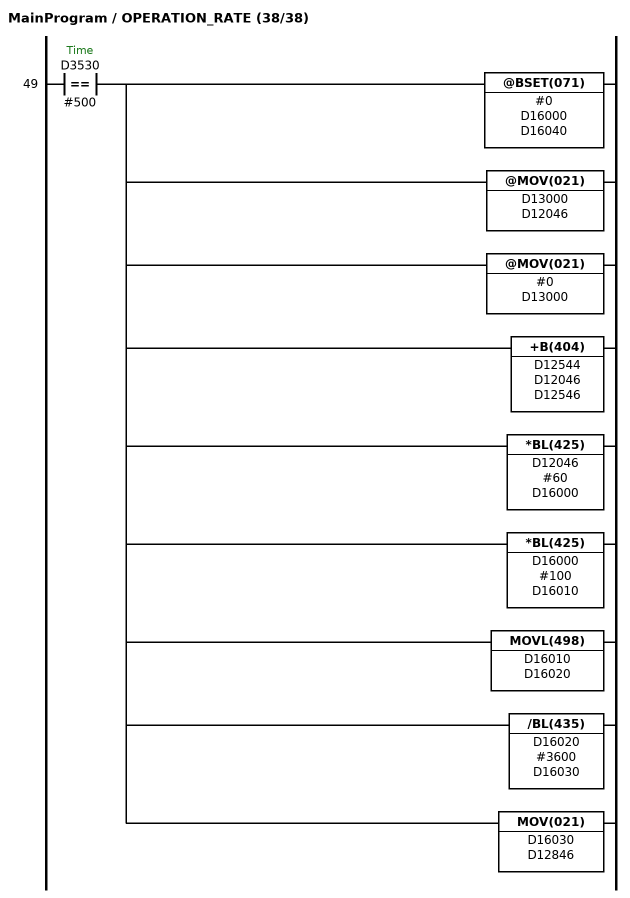
; [picture p288: MainProgram / OPERATION_RATE, rungs 49-49]
; rung 49
LD=L(301) D3530 #500  ; Time
@BSET(071) #0 D16000 D16040
@MOV(021) D13000 D12046
@MOV(021) #0 D13000
+B(404) D12544 D12046 D12546
*BL(425) D12046 #60 D16000
*BL(425) D16000 #100 D16010
MOVL(498) D16010 D16020
/BL(435) D16020 #3600 D16030
MOV(021) D16030 D12846

### Section MASTER_SWITCH_ON

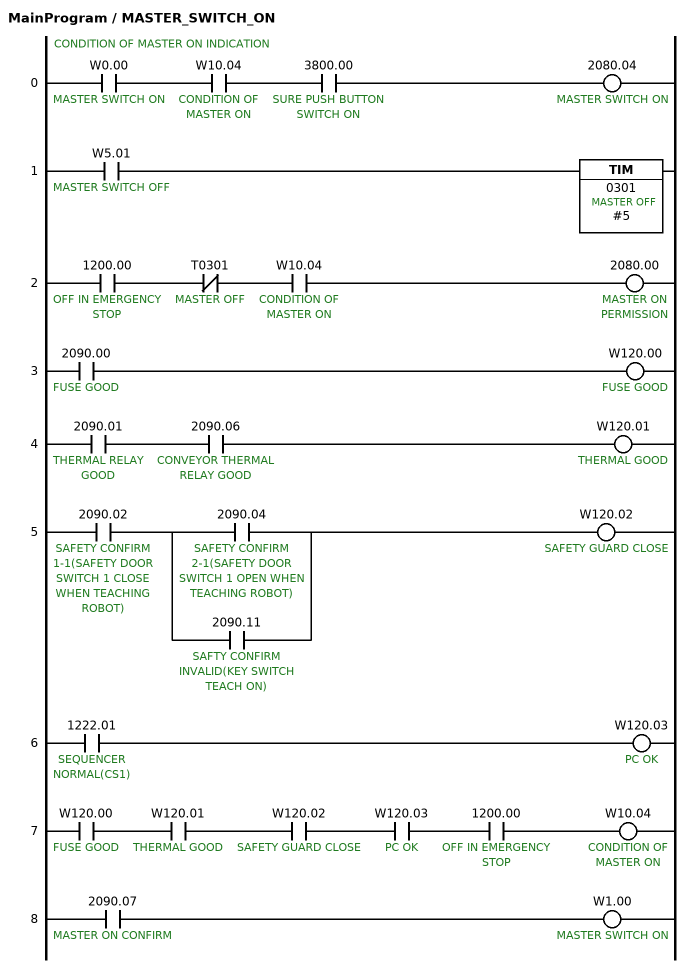
; rung 0: CONDITION OF MASTER ON INDICATION
LD W0.00  ; MASTER SWITCH ON
AND W10.04  ; CONDITION OF MASTER ON
AND 3800.00  ; SURE PUSH BUTTON SWITCH ON
OUT 2080.04  ; MASTER SWITCH ON
; rung 1
LD W5.01  ; MASTER SWITCH OFF
TIM 0301 #5  ; MASTER OFF
; rung 2
LD 1200.00  ; OFF IN EMERGENCY STOP
ANDNOT T0301  ; MASTER OFF
AND W10.04  ; CONDITION OF MASTER ON
OUT 2080.00  ; MASTER ON PERMISSION
; rung 3
LD 2090.00  ; FUSE GOOD
OUT W120.00  ; FUSE GOOD
; rung 4
LD 2090.01  ; THERMAL RELAY GOOD
AND 2090.06  ; CONVEYOR THERMAL RELAY GOOD
OUT W120.01  ; THERMAL GOOD
; rung 5
LD 2090.02  ; SAFETY CONFIRM 1-1(SAFETY DOOR SWITCH 1 CLOSE WHEN TEACHING ROBOT)
LD 2090.04  ; SAFETY CONFIRM 2-1(SAFETY DOOR SWITCH 1 OPEN WHEN TEACHING ROBOT)
OR 2090.11  ; SAFTY CONFIRM INVALID(KEY SWITCH TEACH ON)
ANDLD
OUT W120.02  ; SAFETY GUARD CLOSE
; rung 6
LD 1222.01  ; SEQUENCER NORMAL(CS1)
OUT W120.03  ; PC OK
; rung 7
LD W120.00  ; FUSE GOOD
AND W120.01  ; THERMAL GOOD
AND W120.02  ; SAFETY GUARD CLOSE
AND W120.03  ; PC OK
AND 1200.00  ; OFF IN EMERGENCY STOP
OUT W10.04  ; CONDITION OF MASTER ON
; rung 8
LD 2090.07  ; MASTER ON CONFIRM
OUT W1.00  ; MASTER SWITCH ON

### Section MODE_SELECT

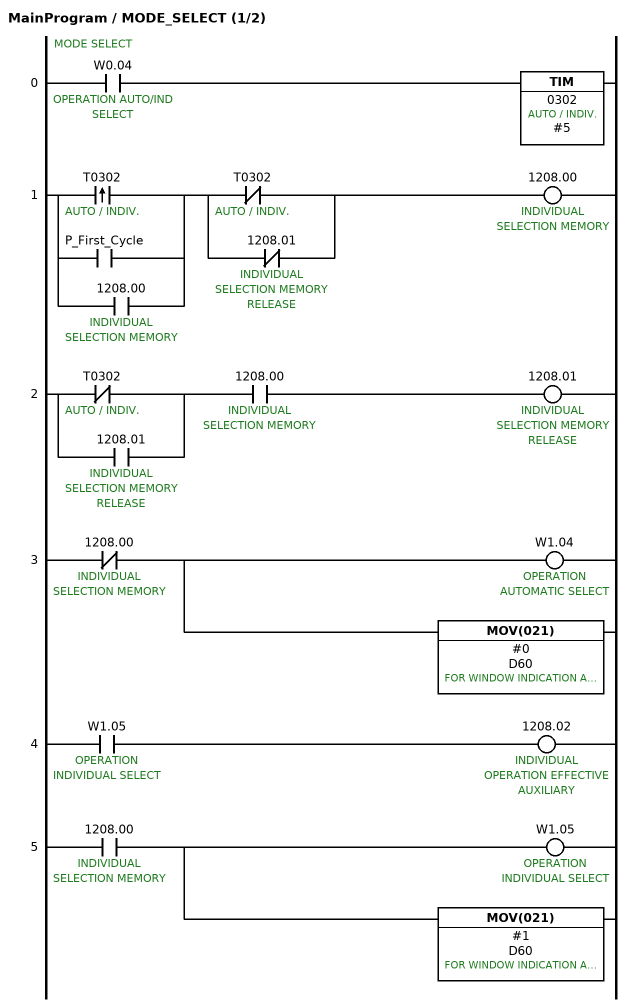
; rung 0: MODE SELECT
LD W0.04  ; OPERATION AUTO/IND SELECT
TIM 0302 #5  ; AUTO / INDIV.
; rung 1
@LD T0302  ; AUTO / INDIV.
OR P_First_Cycle
OR 1208.00  ; INDIVIDUAL SELECTION MEMORY
LDNOT T0302  ; AUTO / INDIV.
ORNOT 1208.01  ; INDIVIDUAL SELECTION MEMORY RELEASE
ANDLD
OUT 1208.00  ; INDIVIDUAL SELECTION MEMORY
; rung 2
LDNOT T0302  ; AUTO / INDIV.
OR 1208.01  ; INDIVIDUAL SELECTION MEMORY RELEASE
AND 1208.00  ; INDIVIDUAL SELECTION MEMORY
OUT 1208.01  ; INDIVIDUAL SELECTION MEMORY RELEASE
; rung 3
LDNOT 1208.00  ; INDIVIDUAL SELECTION MEMORY
OUT W1.04  ; OPERATION AUTOMATIC SELECT
MOV(021) #0 D60  ; FOR WINDOW INDICATION AT INDIVIDUAL
; rung 4
LD W1.05  ; OPERATION INDIVIDUAL SELECT
OUT 1208.02  ; INDIVIDUAL OPERATION EFFECTIVE AUXILIARY
; rung 5
LD 1208.00  ; INDIVIDUAL SELECTION MEMORY
OUT W1.05  ; OPERATION INDIVIDUAL SELECT
MOV(021) #1 D60  ; FOR WINDOW INDICATION AT INDIVIDUAL

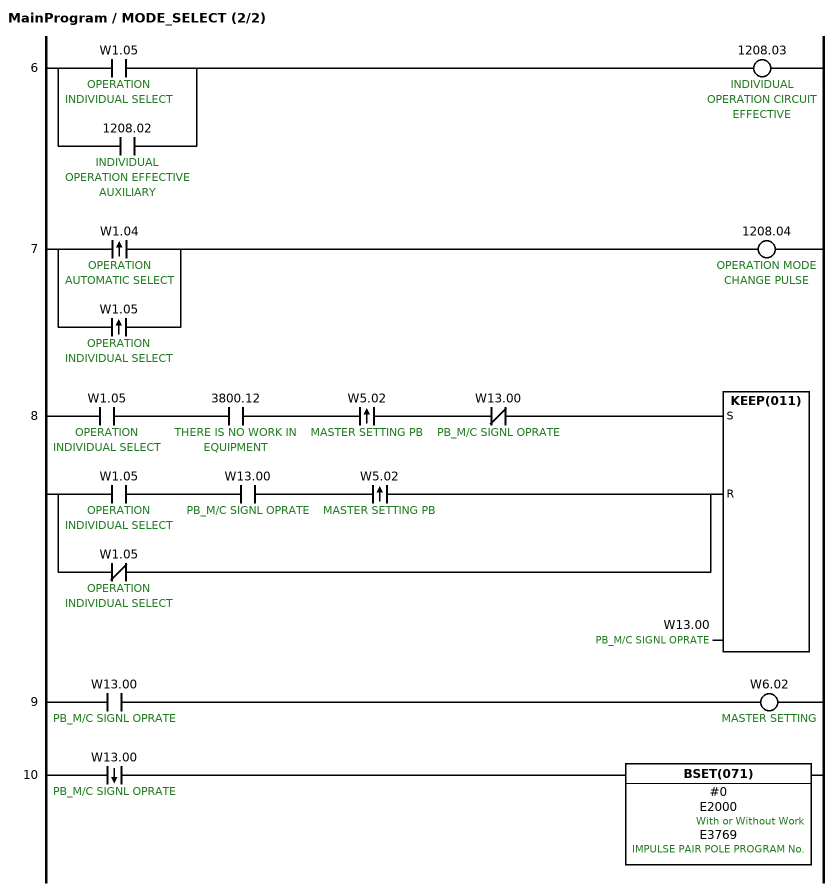
; rung 6
LD W1.05  ; OPERATION INDIVIDUAL SELECT
OR 1208.02  ; INDIVIDUAL OPERATION EFFECTIVE AUXILIARY
OUT 1208.03  ; INDIVIDUAL OPERATION CIRCUIT EFFECTIVE
; rung 7
@LD W1.04  ; OPERATION AUTOMATIC SELECT
@OR W1.05  ; OPERATION INDIVIDUAL SELECT
OUT 1208.04  ; OPERATION MODE CHANGE PULSE
; rung 8
LD W1.05  ; OPERATION INDIVIDUAL SELECT
AND 3800.12  ; THERE IS NO WORK IN EQUIPMENT
@AND W5.02  ; MASTER SETTING PB
ANDNOT W13.00  ; PB_M/C SIGNL OPRATE
LD W1.05  ; OPERATION INDIVIDUAL SELECT
AND W13.00  ; PB_M/C SIGNL OPRATE
@AND W5.02  ; MASTER SETTING PB
ORNOT W1.05  ; OPERATION INDIVIDUAL SELECT
KEEP(011) W13.00  ; PB_M/C SIGNL OPRATE
; rung 9
LD W13.00  ; PB_M/C SIGNL OPRATE
OUT W6.02  ; MASTER SETTING
; rung 10
%LD W13.00  ; PB_M/C SIGNL OPRATE
BSET(071) #0 E2000 E3769  ; With or Without Work, IMPULSE PAIR POLE PROGRAM No.

### Section AUTO_START

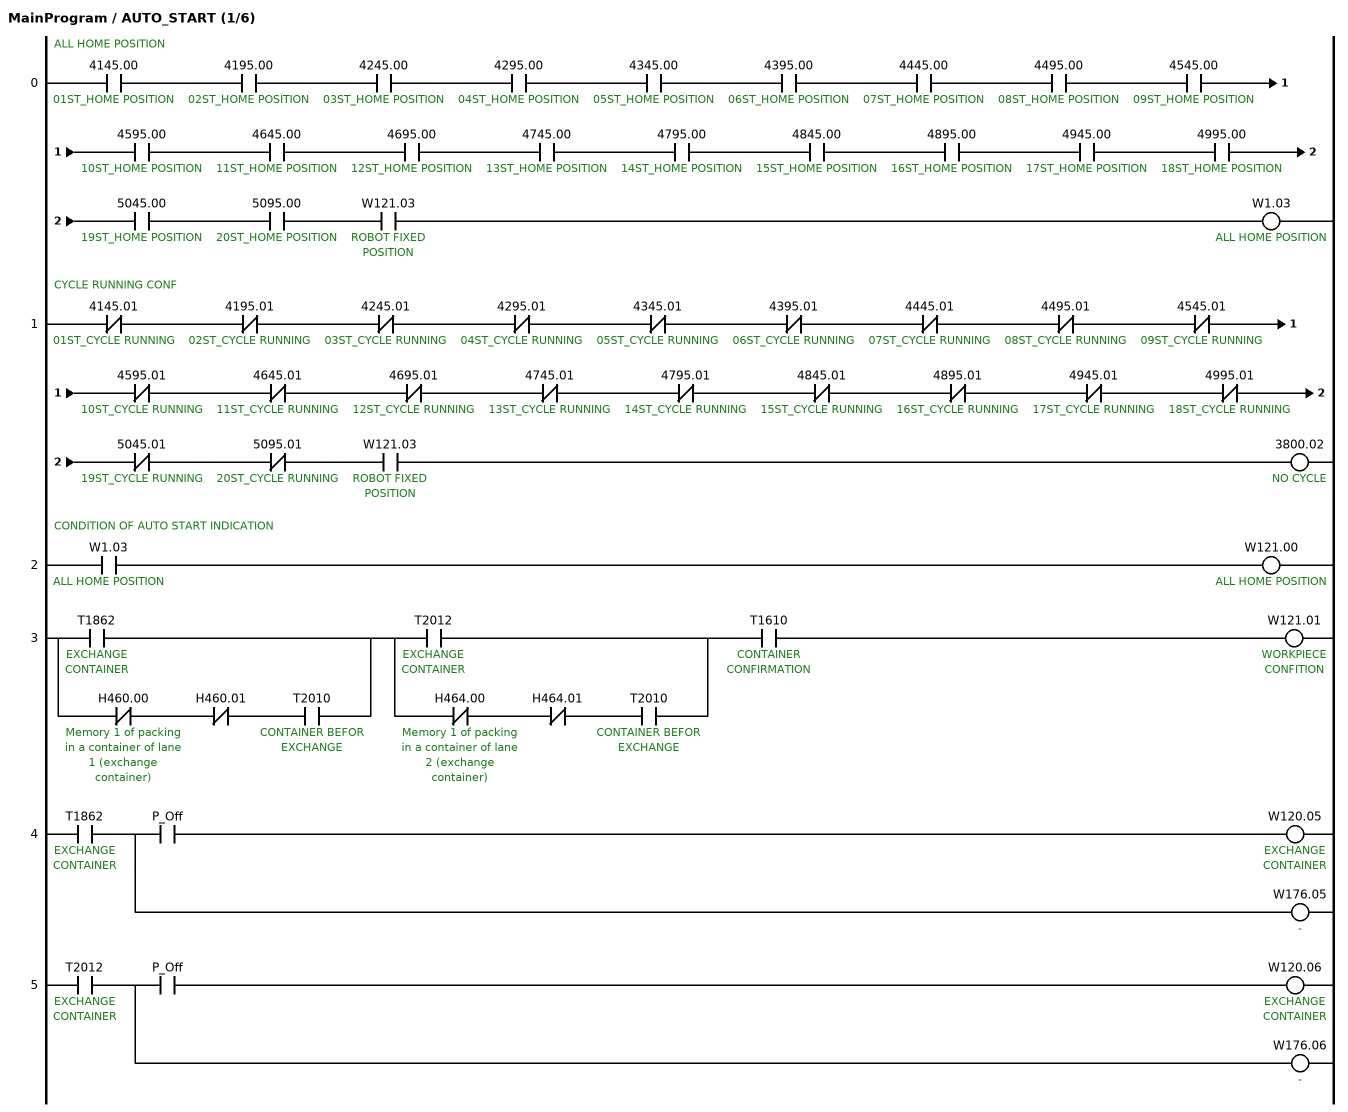
; rung 0: ALL HOME POSITION
LD 4145.00  ; 01ST_HOME POSITION
AND 4195.00  ; 02ST_HOME POSITION
AND 4245.00  ; 03ST_HOME POSITION
AND 4295.00  ; 04ST_HOME POSITION
AND 4345.00  ; 05ST_HOME POSITION
AND 4395.00  ; 06ST_HOME POSITION
AND 4445.00  ; 07ST_HOME POSITION
AND 4495.00  ; 08ST_HOME POSITION
AND 4545.00  ; 09ST_HOME POSITION
AND 4595.00  ; 10ST_HOME POSITION
AND 4645.00  ; 11ST_HOME POSITION
AND 4695.00  ; 12ST_HOME POSITION
AND 4745.00  ; 13ST_HOME POSITION
AND 4795.00  ; 14ST_HOME POSITION
AND 4845.00  ; 15ST_HOME POSITION
AND 4895.00  ; 16ST_HOME POSITION
AND 4945.00  ; 17ST_HOME POSITION
AND 4995.00  ; 18ST_HOME POSITION
AND 5045.00  ; 19ST_HOME POSITION
AND 5095.00  ; 20ST_HOME POSITION
AND W121.03  ; ROBOT FIXED POSITION
OUT W1.03  ; ALL HOME POSITION
; rung 1: CYCLE RUNNING CONF
LDNOT 4145.01  ; 01ST_CYCLE RUNNING
ANDNOT 4195.01  ; 02ST_CYCLE RUNNING
ANDNOT 4245.01  ; 03ST_CYCLE RUNNING
ANDNOT 4295.01  ; 04ST_CYCLE RUNNING
ANDNOT 4345.01  ; 05ST_CYCLE RUNNING
ANDNOT 4395.01  ; 06ST_CYCLE RUNNING
ANDNOT 4445.01  ; 07ST_CYCLE RUNNING
ANDNOT 4495.01  ; 08ST_CYCLE RUNNING
ANDNOT 4545.01  ; 09ST_CYCLE RUNNING
ANDNOT 4595.01  ; 10ST_CYCLE RUNNING
ANDNOT 4645.01  ; 11ST_CYCLE RUNNING
ANDNOT 4695.01  ; 12ST_CYCLE RUNNING
ANDNOT 4745.01  ; 13ST_CYCLE RUNNING
ANDNOT 4795.01  ; 14ST_CYCLE RUNNING
ANDNOT 4845.01  ; 15ST_CYCLE RUNNING
ANDNOT 4895.01  ; 16ST_CYCLE RUNNING
ANDNOT 4945.01  ; 17ST_CYCLE RUNNING
ANDNOT 4995.01  ; 18ST_CYCLE RUNNING
ANDNOT 5045.01  ; 19ST_CYCLE RUNNING
ANDNOT 5095.01  ; 20ST_CYCLE RUNNING
AND W121.03  ; ROBOT FIXED POSITION
OUT 3800.02  ; NO CYCLE
; rung 2: CONDITION OF AUTO START INDICATION
LD W1.03  ; ALL HOME POSITION
OUT W121.00  ; ALL HOME POSITION
; rung 3
LD T1862  ; EXCHANGE CONTAINER
LDNOT H460.00  ; Memory 1 of packing in a container of lane 1 (exchange container)
ANDNOT H460.01
AND T2010  ; CONTAINER BEFOR EXCHANGE
ORLD
LD T2012  ; EXCHANGE CONTAINER
LDNOT H464.00  ; Memory 1 of packing in a container of lane 2 (exchange container)
ANDNOT H464.01
AND T2010  ; CONTAINER BEFOR EXCHANGE
ORLD
ANDLD
AND T1610  ; CONTAINER CONFIRMATION
OUT W121.01  ; WORKPIECE CONFITION
; rung 4
LD T1862  ; EXCHANGE CONTAINER
OUT TR0
AND P_Off
OUT W120.05  ; EXCHANGE CONTAINER
LD TR0
OUT W176.05  ; -
; rung 5
LD T2012  ; EXCHANGE CONTAINER
OUT TR0
AND P_Off
OUT W120.06  ; EXCHANGE CONTAINER
LD TR0
OUT W176.06  ; -

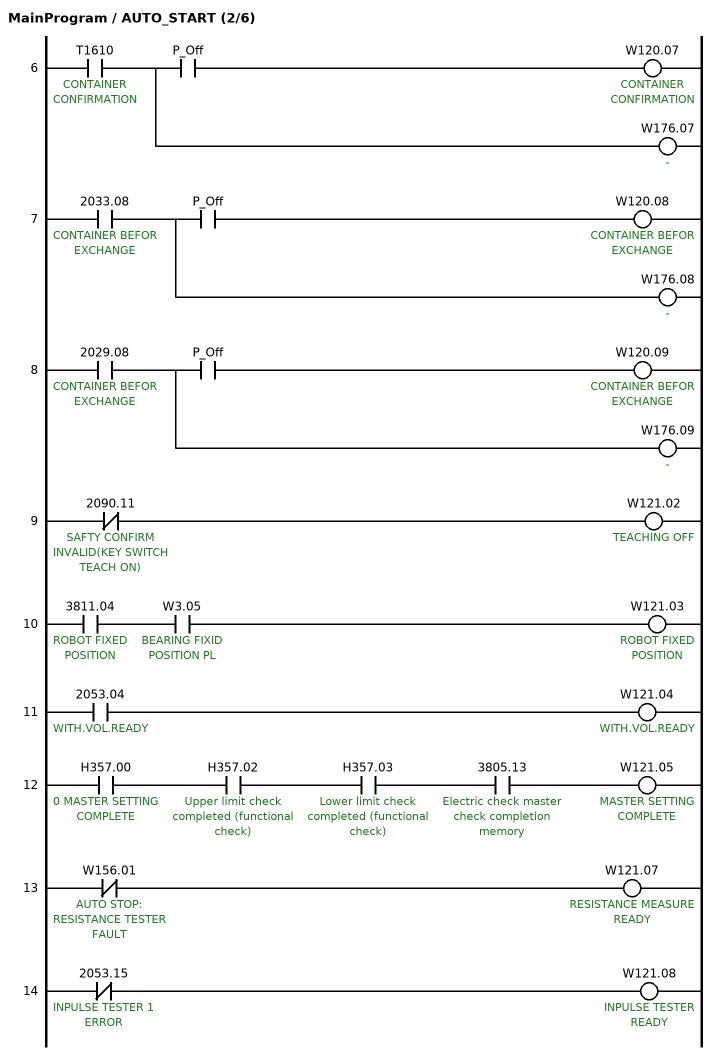
; rung 6
LD T1610  ; CONTAINER CONFIRMATION
OUT TR0
AND P_Off
OUT W120.07  ; CONTAINER CONFIRMATION
LD TR0
OUT W176.07  ; -
; rung 7
LD 2033.08  ; CONTAINER BEFOR EXCHANGE
OUT TR0
AND P_Off
OUT W120.08  ; CONTAINER BEFOR EXCHANGE
LD TR0
OUT W176.08  ; -
; rung 8
LD 2029.08  ; CONTAINER BEFOR EXCHANGE
OUT TR0
AND P_Off
OUT W120.09  ; CONTAINER BEFOR EXCHANGE
LD TR0
OUT W176.09  ; -
; rung 9
LDNOT 2090.11  ; SAFTY CONFIRM INVALID(KEY SWITCH TEACH ON)
OUT W121.02  ; TEACHING OFF
; rung 10
LD 3811.04  ; ROBOT FIXED POSITION
AND W3.05  ; BEARING FIXID POSITION PL
OUT W121.03  ; ROBOT FIXED POSITION
; rung 11
LD 2053.04  ; WITH.VOL.READY
OUT W121.04  ; WITH.VOL.READY
; rung 12
LD H357.00  ; 0 MASTER SETTING COMPLETE
AND H357.02  ; Upper limit check completed (functional check)
AND H357.03  ; Lower limit check completed (functional check)
AND 3805.13  ; Electric check master check completion memory
OUT W121.05  ; MASTER SETTING COMPLETE
; rung 13
LDNOT W156.01  ; AUTO STOP:RESISTANCE TESTER FAULT
OUT W121.07  ; RESISTANCE MEASURE READY
; rung 14
LDNOT 2053.15  ; INPULSE TESTER 1 ERROR
OUT W121.08  ; INPULSE TESTER READY

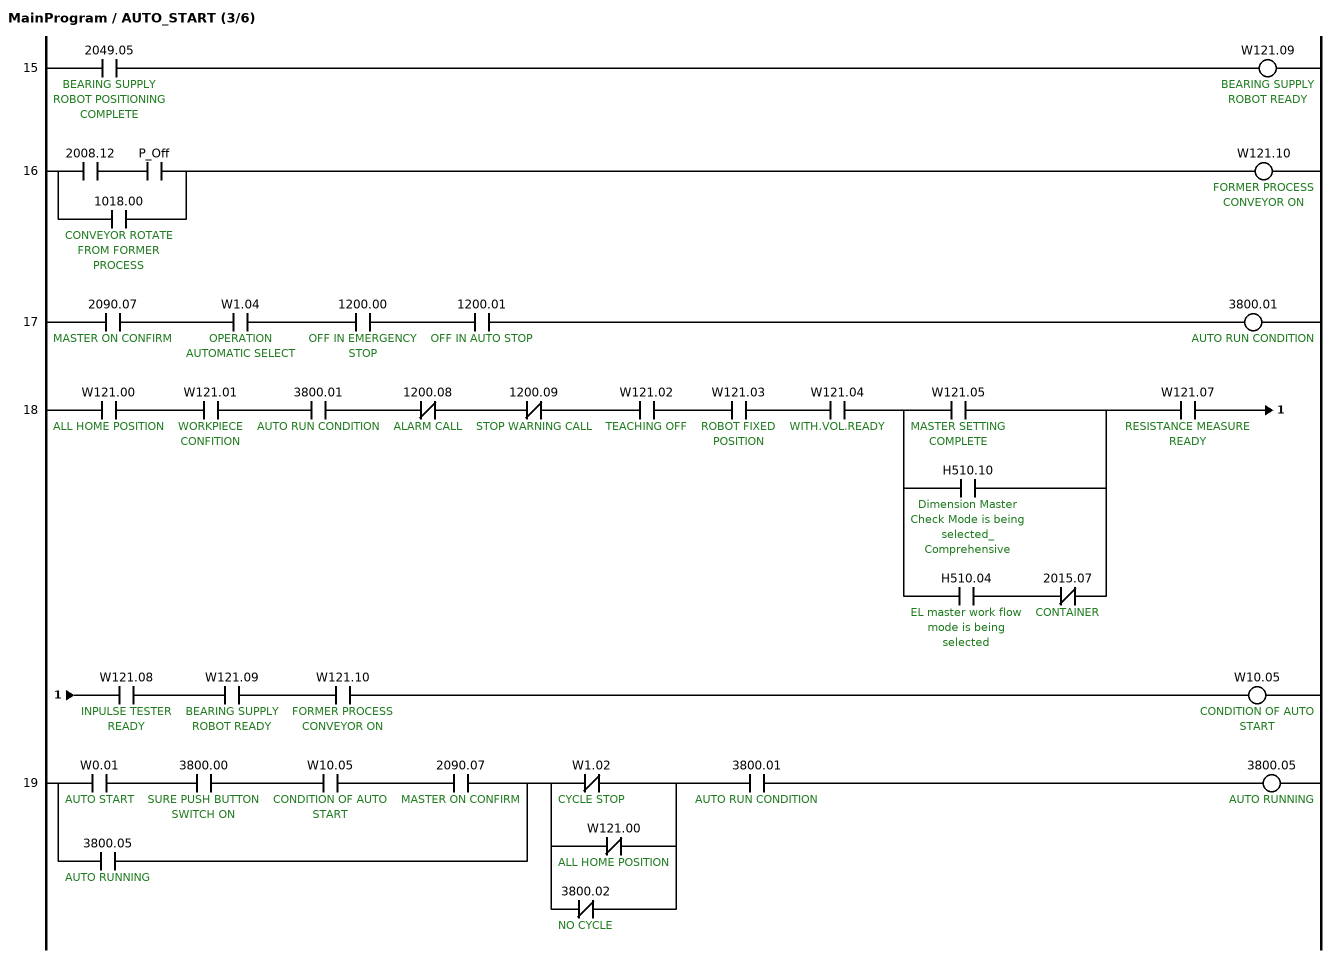
; rung 15
LD 2049.05  ; BEARING SUPPLY ROBOT POSITIONING COMPLETE
OUT W121.09  ; BEARING SUPPLY ROBOT READY
; rung 16
LD 2008.12
AND P_Off
OR 1018.00  ; CONVEYOR ROTATE FROM FORMER PROCESS
OUT W121.10  ; FORMER PROCESS CONVEYOR ON
; rung 17
LD 2090.07  ; MASTER ON CONFIRM
AND W1.04  ; OPERATION AUTOMATIC SELECT
AND 1200.00  ; OFF IN EMERGENCY STOP
AND 1200.01  ; OFF IN AUTO STOP
OUT 3800.01  ; AUTO RUN CONDITION
; rung 18
LD W121.00  ; ALL HOME POSITION
AND W121.01  ; WORKPIECE CONFITION
AND 3800.01  ; AUTO RUN CONDITION
ANDNOT 1200.08  ; ALARM CALL
ANDNOT 1200.09  ; STOP WARNING CALL
AND W121.02  ; TEACHING OFF
AND W121.03  ; ROBOT FIXED POSITION
AND W121.04  ; WITH.VOL.READY
LD W121.05  ; MASTER SETTING COMPLETE
OR H510.10  ; Dimension Master Check Mode is being selected_Comprehensive
LD H510.04  ; EL master work flow mode is being selected
ANDNOT 2015.07  ; CONTAINER
ORLD
ANDLD
AND W121.07  ; RESISTANCE MEASURE READY
AND W121.08  ; INPULSE TESTER READY
AND W121.09  ; BEARING SUPPLY ROBOT READY
AND W121.10  ; FORMER PROCESS CONVEYOR ON
OUT W10.05  ; CONDITION OF AUTO START
; rung 19
LD W0.01  ; AUTO START
AND 3800.00  ; SURE PUSH BUTTON SWITCH ON
AND W10.05  ; CONDITION OF AUTO START
AND 2090.07  ; MASTER ON CONFIRM
OR 3800.05  ; AUTO RUNNING
LDNOT W1.02  ; CYCLE STOP
ORNOT W121.00  ; ALL HOME POSITION
ORNOT 3800.02  ; NO CYCLE
ANDLD
AND 3800.01  ; AUTO RUN CONDITION
OUT 3800.05  ; AUTO RUNNING

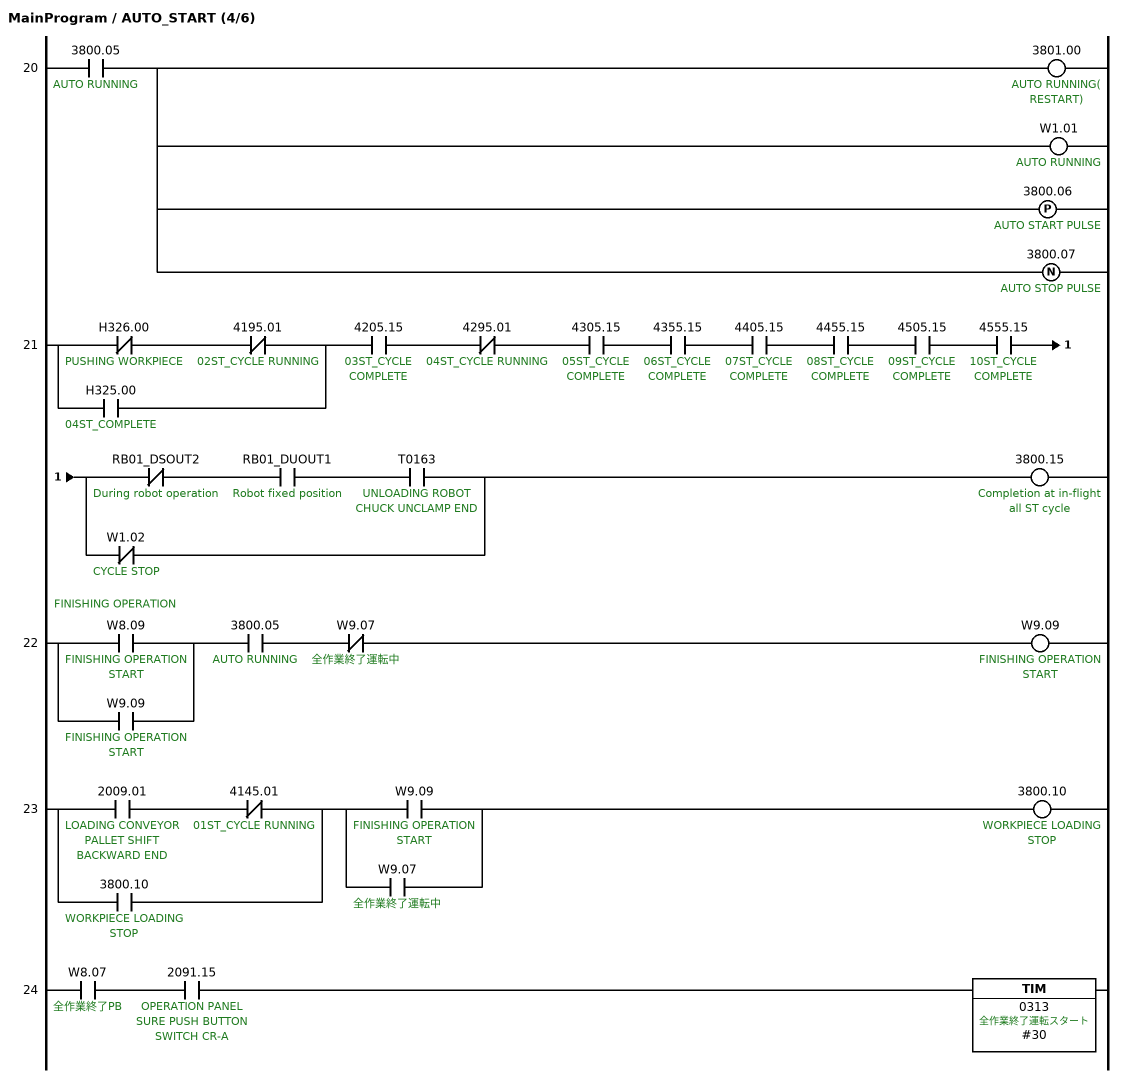
; rung 20
LD 3800.05  ; AUTO RUNNING
OUT 3801.00  ; AUTO RUNNING(RESTART)
OUT W1.01  ; AUTO RUNNING
DIFU(013) 3800.06  ; AUTO START PULSE
DIFD(014) 3800.07  ; AUTO STOP PULSE
; rung 21
LDNOT H326.00  ; PUSHING WORKPIECE
ANDNOT 4195.01  ; 02ST_CYCLE RUNNING
OR H325.00  ; 04ST_COMPLETE
AND 4205.15  ; 03ST_CYCLE COMPLETE
ANDNOT 4295.01  ; 04ST_CYCLE RUNNING
AND 4305.15  ; 05ST_CYCLE COMPLETE
AND 4355.15  ; 06ST_CYCLE COMPLETE
AND 4405.15  ; 07ST_CYCLE COMPLETE
AND 4455.15  ; 08ST_CYCLE COMPLETE
AND 4505.15  ; 09ST_CYCLE COMPLETE
AND 4555.15  ; 10ST_CYCLE COMPLETE
LDNOT RB01_DSOUT2  ; During robot operation
AND RB01_DUOUT1  ; Robot fixed position
AND T0163  ; UNLOADING ROBOT CHUCK UNCLAMP END
ORNOT W1.02  ; CYCLE STOP
ANDLD
OUT 3800.15  ; Completion at in-flight all ST cycle
; rung 22: FINISHING OPERATION
LD W8.09  ; FINISHING OPERATION START
OR W9.09  ; FINISHING OPERATION START
AND 3800.05  ; AUTO RUNNING
ANDNOT W9.07  ; 全作業終了運転中
OUT W9.09  ; FINISHING OPERATION START
; rung 23
LD 2009.01  ; LOADING CONVEYOR PALLET SHIFT BACKWARD END
ANDNOT 4145.01  ; 01ST_CYCLE RUNNING
OR 3800.10  ; WORKPIECE LOADING STOP
LD W9.09  ; FINISHING OPERATION START
OR W9.07  ; 全作業終了運転中
ANDLD
OUT 3800.10  ; WORKPIECE LOADING STOP
; rung 24
LD W8.07  ; 全作業終了PB
AND 2091.15  ; OPERATION PANEL SURE PUSH BUTTON SWITCH CR-A
TIM 0313 #30  ; 全作業終了運転スタート

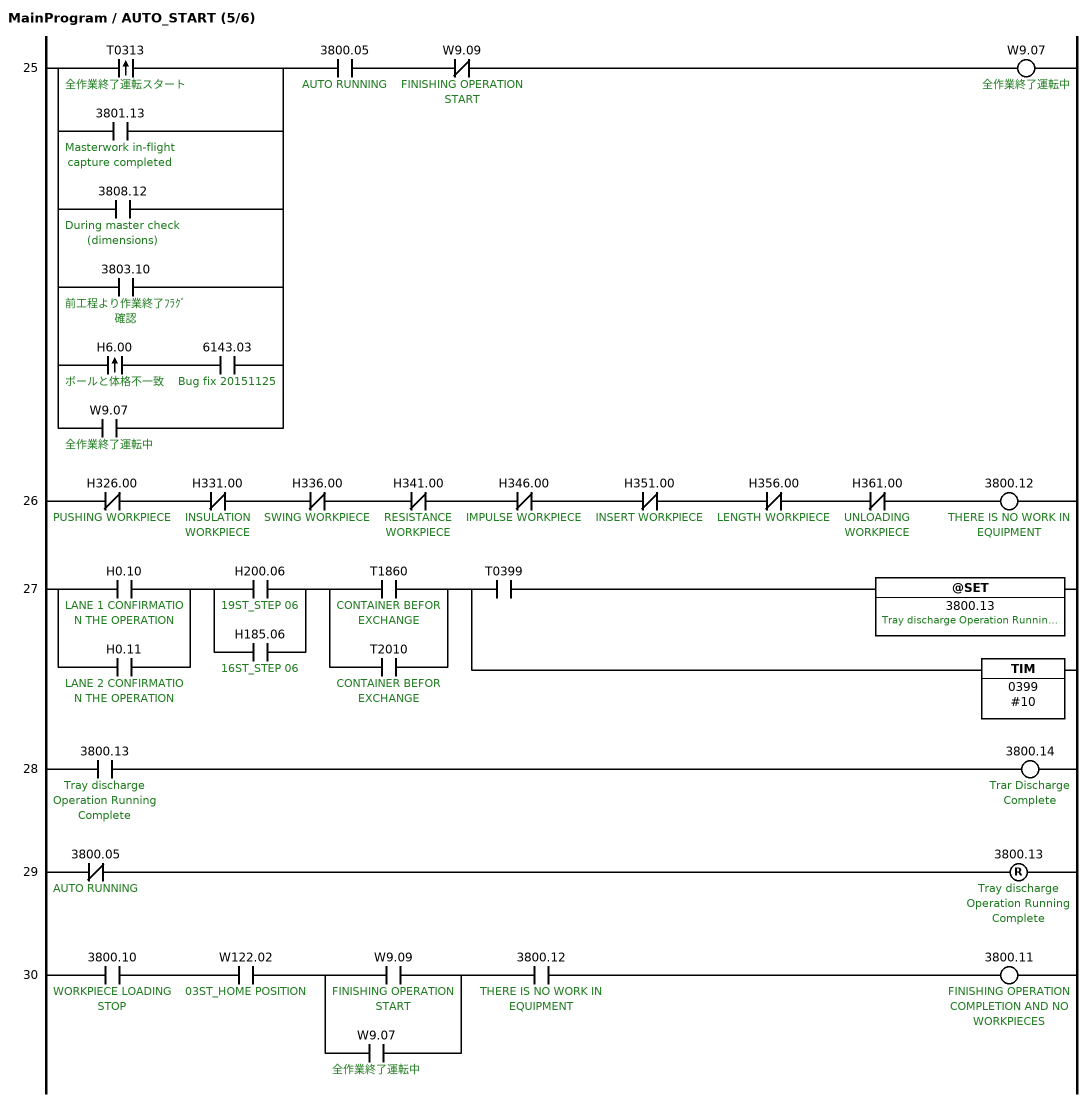
; rung 25
@LD T0313  ; 全作業終了運転スタート
OR 3801.13  ; Masterwork in-flight capture completed
OR 3808.12  ; During master check (dimensions)
OR 3803.10  ; 前工程より作業終了ﾌﾗｸﾞ確認
@LD H6.00  ; ボールと体格不一致
AND 6143.03  ; Bug fix 20151125
ORLD
OR W9.07  ; 全作業終了運転中
AND 3800.05  ; AUTO RUNNING
ANDNOT W9.09  ; FINISHING OPERATION START
OUT W9.07  ; 全作業終了運転中
; rung 26
LDNOT H326.00  ; PUSHING WORKPIECE
ANDNOT H331.00  ; INSULATION WORKPIECE
ANDNOT H336.00  ; SWING WORKPIECE
ANDNOT H341.00  ; RESISTANCE WORKPIECE
ANDNOT H346.00  ; IMPULSE WORKPIECE
ANDNOT H351.00  ; INSERT WORKPIECE
ANDNOT H356.00  ; LENGTH WORKPIECE
ANDNOT H361.00  ; UNLOADING WORKPIECE
OUT 3800.12  ; THERE IS NO WORK IN EQUIPMENT
; rung 27
LD H0.10  ; LANE 1 CONFIRMATION THE OPERATION
OR H0.11  ; LANE 2 CONFIRMATION THE OPERATION
LD H200.06  ; 19ST_STEP 06
OR H185.06  ; 16ST_STEP 06
ANDLD
LD T1860  ; CONTAINER BEFOR EXCHANGE
OR T2010  ; CONTAINER BEFOR EXCHANGE
ANDLD
OUT TR0
AND T0399
@SET 3800.13  ; Tray discharge Operation Running Complete
LD TR0
TIM 0399 #10
; rung 28
LD 3800.13  ; Tray discharge Operation Running Complete
OUT 3800.14  ; Trar Discharge Complete
; rung 29
LDNOT 3800.05  ; AUTO RUNNING
RSET 3800.13  ; Tray discharge Operation Running Complete
; rung 30
LD 3800.10  ; WORKPIECE LOADING STOP
AND W122.02  ; 03ST_HOME POSITION
LD W9.09  ; FINISHING OPERATION START
OR W9.07  ; 全作業終了運転中
ANDLD
AND 3800.12  ; THERE IS NO WORK IN EQUIPMENT
OUT 3800.11  ; FINISHING OPERATION COMPLETION AND NO WORKPIECES

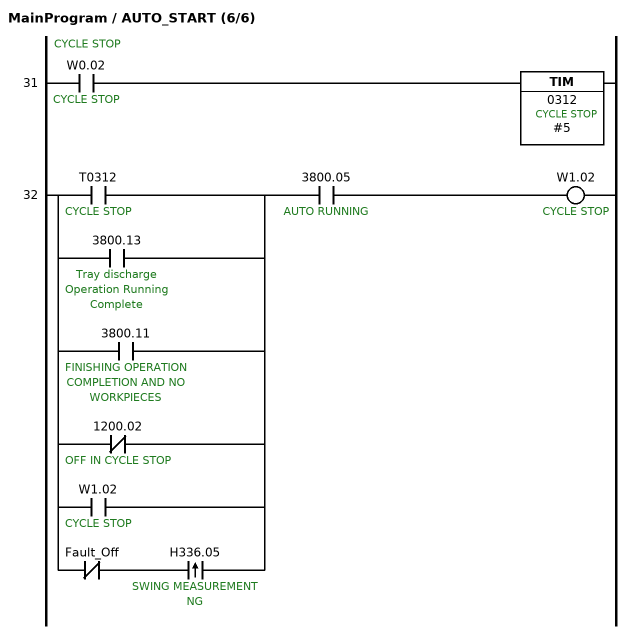
; rung 31: CYCLE STOP
LD W0.02  ; CYCLE STOP
TIM 0312 #5  ; CYCLE STOP
; rung 32
LD T0312  ; CYCLE STOP
OR 3800.13  ; Tray discharge Operation Running Complete
OR 3800.11  ; FINISHING OPERATION COMPLETION AND NO WORKPIECES
ORNOT 1200.02  ; OFF IN CYCLE STOP
OR W1.02  ; CYCLE STOP
LDNOT Fault_Off
@AND H336.05  ; SWING MEASUREMENT NG
ORLD
AND 3800.05  ; AUTO RUNNING
OUT W1.02  ; CYCLE STOP

### Section ST01_LOADING_CV_UNIT
; rung 0: 01ST_LOADING CV UNIT

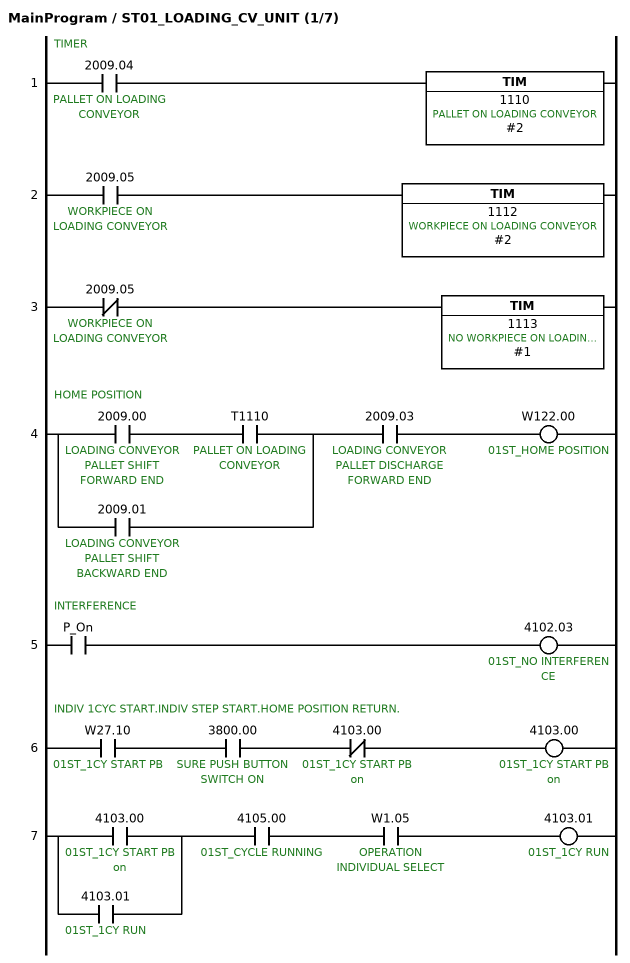
; rung 1: TIMER
LD 2009.04  ; PALLET ON LOADING CONVEYOR
TIM 1110 #2  ; PALLET ON LOADING CONVEYOR
; rung 2
LD 2009.05  ; WORKPIECE ON LOADING CONVEYOR
TIM 1112 #2  ; WORKPIECE ON LOADING CONVEYOR
; rung 3
LDNOT 2009.05  ; WORKPIECE ON LOADING CONVEYOR
TIM 1113 #1  ; NO WORKPIECE ON LOADING CONVEYOR
; rung 4: HOME POSITION
LD 2009.00  ; LOADING CONVEYOR PALLET SHIFT FORWARD END
AND T1110  ; PALLET ON LOADING CONVEYOR
OR 2009.01  ; LOADING CONVEYOR PALLET SHIFT BACKWARD END
AND 2009.03  ; LOADING CONVEYOR PALLET DISCHARGE FORWARD END
OUT W122.00  ; 01ST_HOME POSITION
; rung 5: INTERFERENCE
LD P_On
OUT 4102.03  ; 01ST_NO INTERFERENCE
; rung 6: INDIV 1CYC START.INDIV STEP START.HOME POSITION RETURN.
LD W27.10  ; 01ST_1CY START PB
AND 3800.00  ; SURE PUSH BUTTON SWITCH ON
ANDNOT 4103.00  ; 01ST_1CY START PB on
OUT 4103.00  ; 01ST_1CY START PB on
; rung 7
LD 4103.00  ; 01ST_1CY START PB on
OR 4103.01  ; 01ST_1CY RUN
AND 4105.00  ; 01ST_CYCLE RUNNING
AND W1.05  ; OPERATION INDIVIDUAL SELECT
OUT 4103.01  ; 01ST_1CY RUN

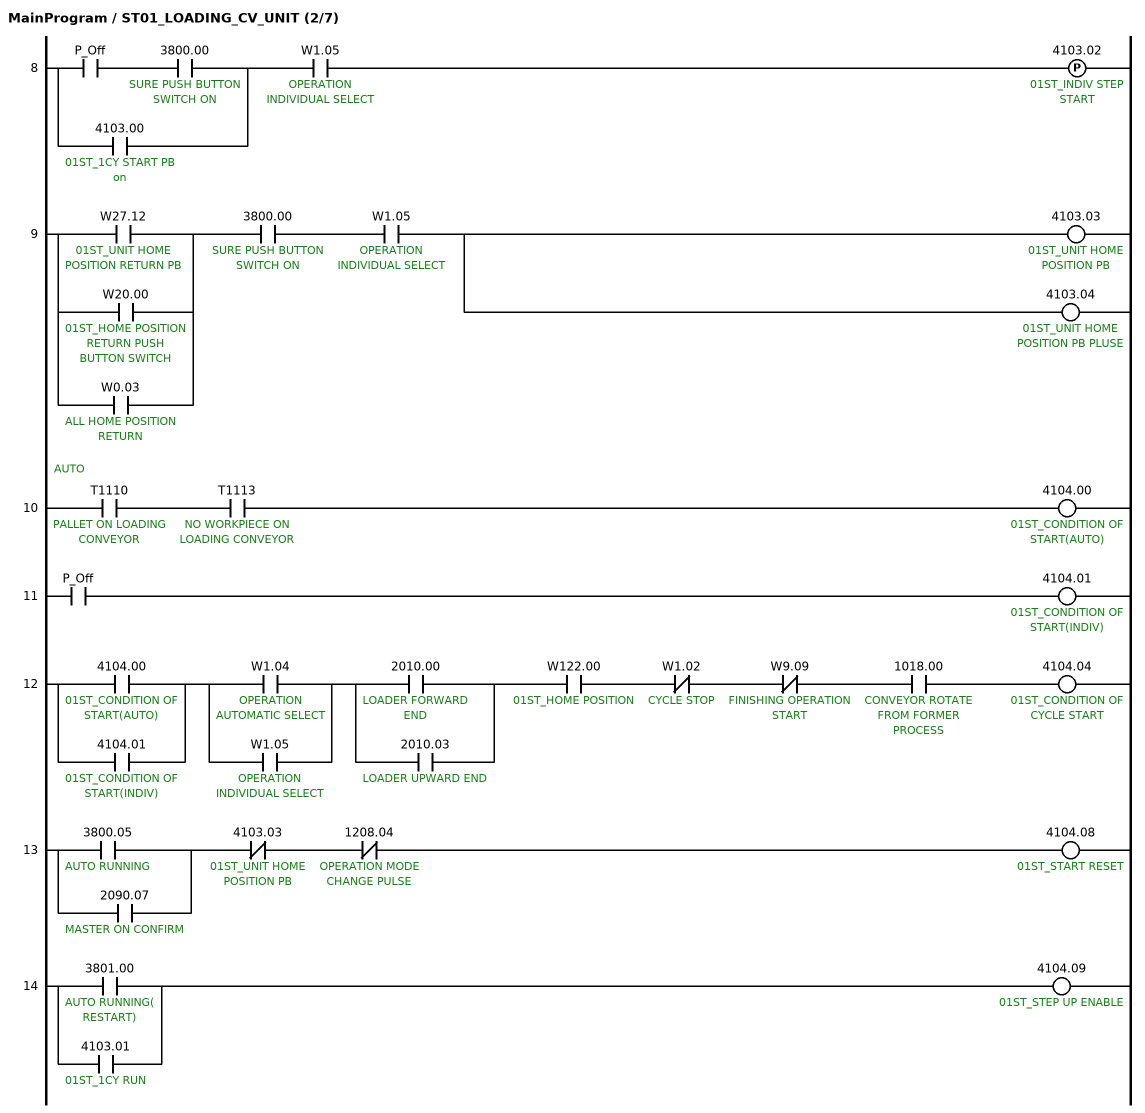
; rung 8
LD P_Off
AND 3800.00  ; SURE PUSH BUTTON SWITCH ON
OR 4103.00  ; 01ST_1CY START PB on
AND W1.05  ; OPERATION INDIVIDUAL SELECT
DIFU(013) 4103.02  ; 01ST_INDIV STEP START
; rung 9
LD W27.12  ; 01ST_UNIT HOME POSITION RETURN PB
OR W20.00  ; 01ST_HOME POSITION RETURN PUSH BUTTON SWITCH
OR W0.03  ; ALL HOME POSITION RETURN
AND 3800.00  ; SURE PUSH BUTTON SWITCH ON
AND W1.05  ; OPERATION INDIVIDUAL SELECT
OUT 4103.03  ; 01ST_UNIT HOME POSITION PB
OUT 4103.04  ; 01ST_UNIT HOME POSITION PB PLUSE
; rung 10: AUTO
LD T1110  ; PALLET ON LOADING CONVEYOR
AND T1113  ; NO WORKPIECE ON LOADING CONVEYOR
OUT 4104.00  ; 01ST_CONDITION OF START(AUTO)
; rung 11
LD P_Off
OUT 4104.01  ; 01ST_CONDITION OF START(INDIV)
; rung 12
LD 4104.00  ; 01ST_CONDITION OF START(AUTO)
OR 4104.01  ; 01ST_CONDITION OF START(INDIV)
LD W1.04  ; OPERATION AUTOMATIC SELECT
OR W1.05  ; OPERATION INDIVIDUAL SELECT
ANDLD
LD 2010.00  ; LOADER FORWARD END
OR 2010.03  ; LOADER UPWARD END
ANDLD
AND W122.00  ; 01ST_HOME POSITION
ANDNOT W1.02  ; CYCLE STOP
ANDNOT W9.09  ; FINISHING OPERATION START
AND 1018.00  ; CONVEYOR ROTATE FROM FORMER PROCESS
OUT 4104.04  ; 01ST_CONDITION OF CYCLE START
; rung 13
LD 3800.05  ; AUTO RUNNING
OR 2090.07  ; MASTER ON CONFIRM
ANDNOT 4103.03  ; 01ST_UNIT HOME POSITION PB
ANDNOT 1208.04  ; OPERATION MODE CHANGE PULSE
OUT 4104.08  ; 01ST_START RESET
; rung 14
LD 3801.00  ; AUTO RUNNING(RESTART)
OR 4103.01  ; 01ST_1CY RUN
OUT 4104.09  ; 01ST_STEP UP ENABLE

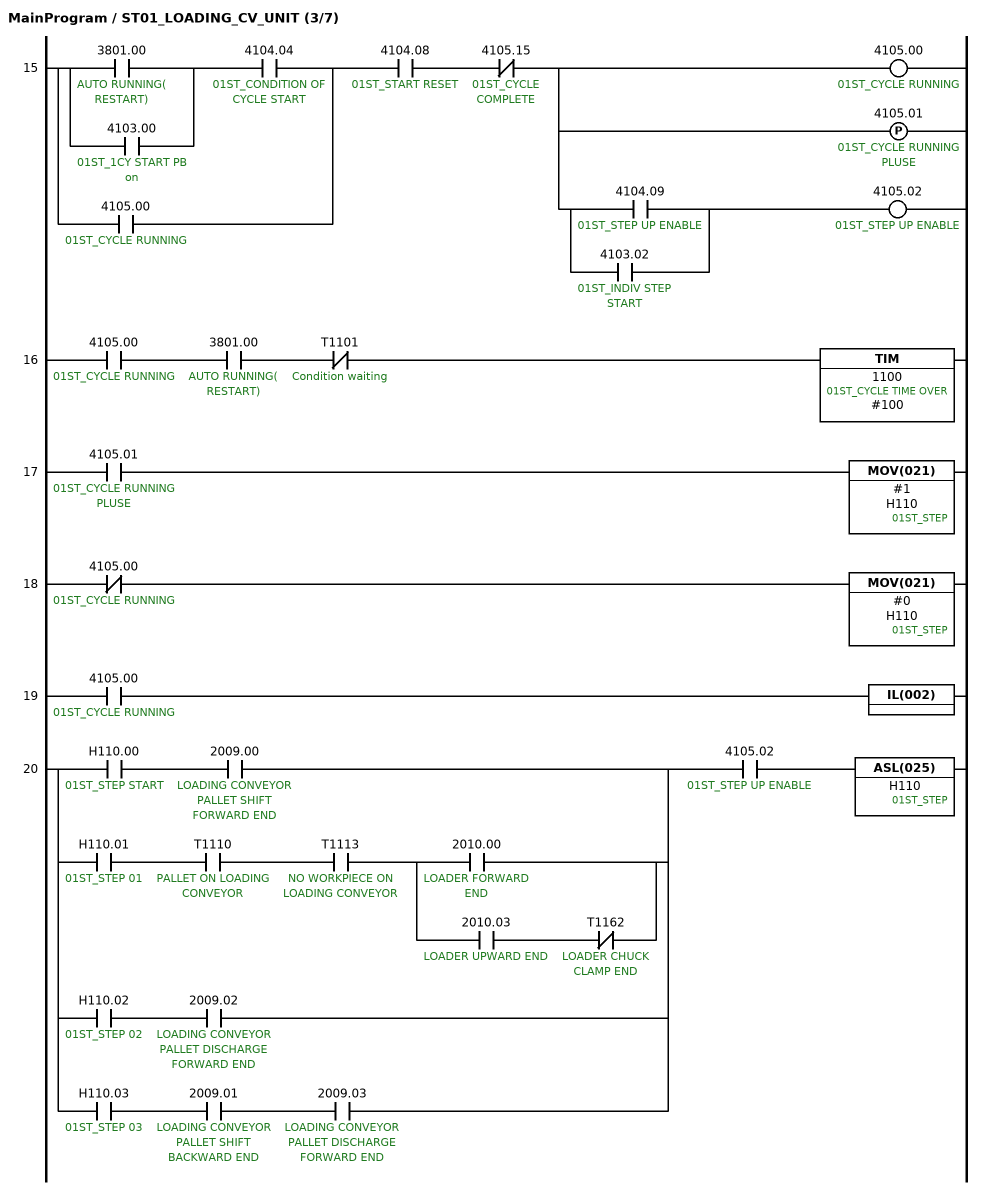
; rung 15
LD 3801.00  ; AUTO RUNNING(RESTART)
OR 4103.00  ; 01ST_1CY START PB on
AND 4104.04  ; 01ST_CONDITION OF CYCLE START
OR 4105.00  ; 01ST_CYCLE RUNNING
AND 4104.08  ; 01ST_START RESET
ANDNOT 4105.15  ; 01ST_CYCLE COMPLETE
OUT 4105.00  ; 01ST_CYCLE RUNNING
DIFU(013) 4105.01  ; 01ST_CYCLE RUNNING PLUSE
LD 4104.09  ; 01ST_STEP UP ENABLE
OR 4103.02  ; 01ST_INDIV STEP START
ANDLD
OUT 4105.02  ; 01ST_STEP UP ENABLE
; rung 16
LD 4105.00  ; 01ST_CYCLE RUNNING
AND 3801.00  ; AUTO RUNNING(RESTART)
ANDNOT T1101  ; Condition waiting
TIM 1100 #100  ; 01ST_CYCLE TIME OVER
; rung 17
LD 4105.01  ; 01ST_CYCLE RUNNING PLUSE
MOV(021) #1 H110  ; 01ST_STEP
; rung 18
LDNOT 4105.00  ; 01ST_CYCLE RUNNING
MOV(021) #0 H110  ; 01ST_STEP
; rung 19
LD 4105.00  ; 01ST_CYCLE RUNNING
IL(002)
; rung 20
LD H110.00  ; 01ST_STEP START
AND 2009.00  ; LOADING CONVEYOR PALLET SHIFT FORWARD END
LD H110.01  ; 01ST_STEP 01
AND T1110  ; PALLET ON LOADING CONVEYOR
AND T1113  ; NO WORKPIECE ON LOADING CONVEYOR
LD 2010.00  ; LOADER FORWARD END
LD 2010.03  ; LOADER UPWARD END
ANDNOT T1162  ; LOADER CHUCK CLAMP END
ORLD
ANDLD
ORLD
LD H110.02  ; 01ST_STEP 02
AND 2009.02  ; LOADING CONVEYOR PALLET DISCHARGE FORWARD END
ORLD
LD H110.03  ; 01ST_STEP 03
AND 2009.01  ; LOADING CONVEYOR PALLET SHIFT BACKWARD END
AND 2009.03  ; LOADING CONVEYOR PALLET DISCHARGE FORWARD END
ORLD
AND 4105.02  ; 01ST_STEP UP ENABLE
ASL(025) H110  ; 01ST_STEP

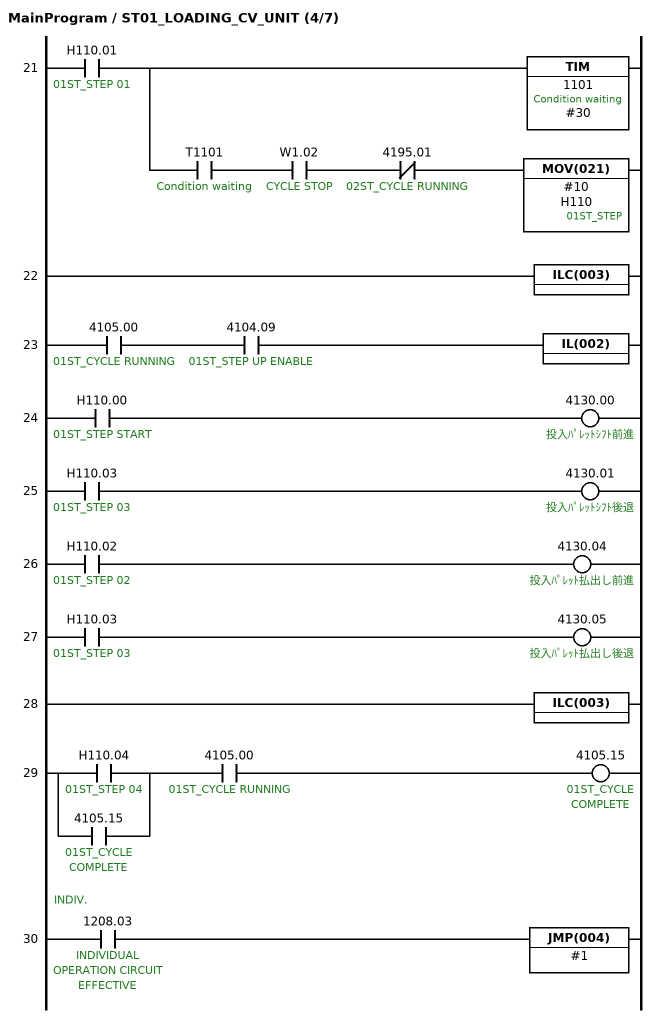
; rung 21
LD H110.01  ; 01ST_STEP 01
TIM 1101 #30  ; Condition waiting
AND T1101  ; Condition waiting
AND W1.02  ; CYCLE STOP
ANDNOT 4195.01  ; 02ST_CYCLE RUNNING
MOV(021) #10 H110  ; 01ST_STEP
; rung 22
ILC(003)
; rung 23
LD 4105.00  ; 01ST_CYCLE RUNNING
AND 4104.09  ; 01ST_STEP UP ENABLE
IL(002)
; rung 24
LD H110.00  ; 01ST_STEP START
OUT 4130.00  ; 投入ﾊﾟﾚｯﾄｼﾌﾄ前進
; rung 25
LD H110.03  ; 01ST_STEP 03
OUT 4130.01  ; 投入ﾊﾟﾚｯﾄｼﾌﾄ後退
; rung 26
LD H110.02  ; 01ST_STEP 02
OUT 4130.04  ; 投入ﾊﾟﾚｯﾄ払出し前進
; rung 27
LD H110.03  ; 01ST_STEP 03
OUT 4130.05  ; 投入ﾊﾟﾚｯﾄ払出し後退
; rung 28
ILC(003)
; rung 29
LD H110.04  ; 01ST_STEP 04
OR 4105.15  ; 01ST_CYCLE COMPLETE
AND 4105.00  ; 01ST_CYCLE RUNNING
OUT 4105.15  ; 01ST_CYCLE COMPLETE
; rung 30: INDIV.
LD 1208.03  ; INDIVIDUAL OPERATION CIRCUIT EFFECTIVE
JMP(004) #1

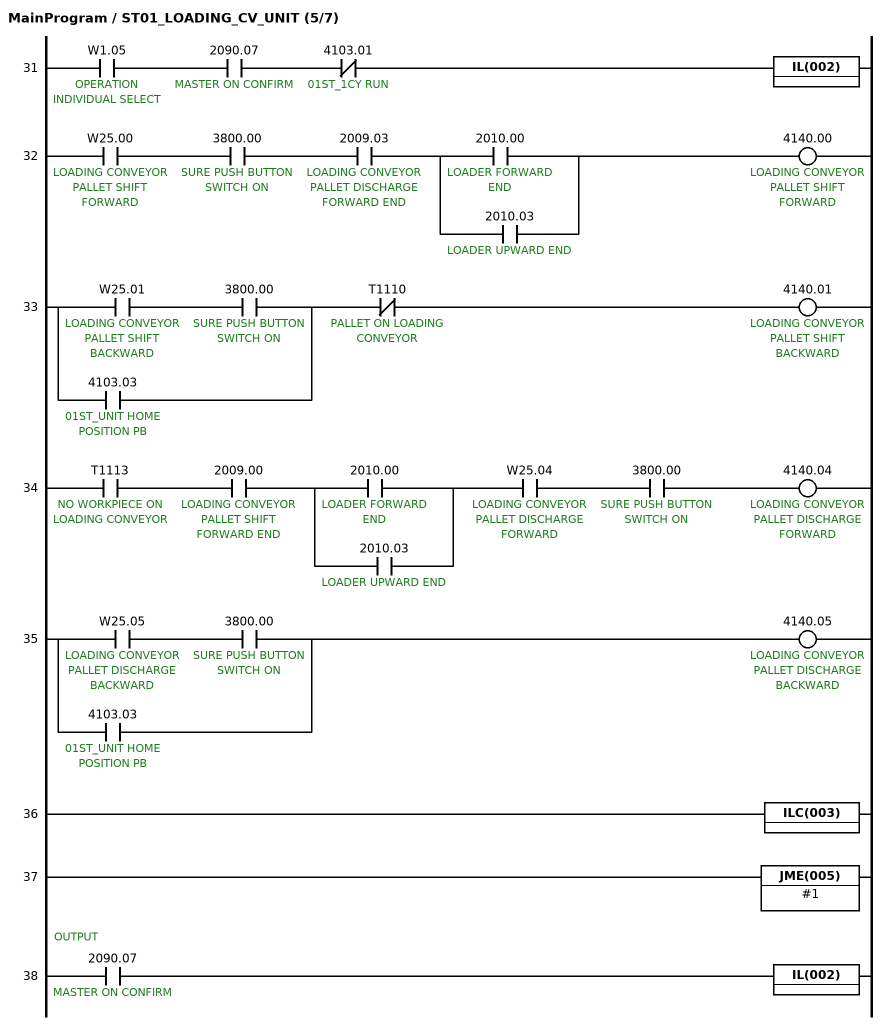
; rung 31
LD W1.05  ; OPERATION INDIVIDUAL SELECT
AND 2090.07  ; MASTER ON CONFIRM
ANDNOT 4103.01  ; 01ST_1CY RUN
IL(002)
; rung 32
LD W25.00  ; LOADING CONVEYOR PALLET SHIFT FORWARD
AND 3800.00  ; SURE PUSH BUTTON SWITCH ON
AND 2009.03  ; LOADING CONVEYOR PALLET DISCHARGE FORWARD END
LD 2010.00  ; LOADER FORWARD END
OR 2010.03  ; LOADER UPWARD END
ANDLD
OUT 4140.00  ; LOADING CONVEYOR PALLET SHIFT FORWARD
; rung 33
LD W25.01  ; LOADING CONVEYOR PALLET SHIFT BACKWARD
AND 3800.00  ; SURE PUSH BUTTON SWITCH ON
OR 4103.03  ; 01ST_UNIT HOME POSITION PB
ANDNOT T1110  ; PALLET ON LOADING CONVEYOR
OUT 4140.01  ; LOADING CONVEYOR PALLET SHIFT BACKWARD
; rung 34
LD T1113  ; NO WORKPIECE ON LOADING CONVEYOR
AND 2009.00  ; LOADING CONVEYOR PALLET SHIFT FORWARD END
LD 2010.00  ; LOADER FORWARD END
OR 2010.03  ; LOADER UPWARD END
ANDLD
AND W25.04  ; LOADING CONVEYOR PALLET DISCHARGE FORWARD
AND 3800.00  ; SURE PUSH BUTTON SWITCH ON
OUT 4140.04  ; LOADING CONVEYOR PALLET DISCHARGE FORWARD
; rung 35
LD W25.05  ; LOADING CONVEYOR PALLET DISCHARGE BACKWARD
AND 3800.00  ; SURE PUSH BUTTON SWITCH ON
OR 4103.03  ; 01ST_UNIT HOME POSITION PB
OUT 4140.05  ; LOADING CONVEYOR PALLET DISCHARGE BACKWARD
; rung 36
ILC(003)
; rung 37
JME(005) #1
; rung 38: OUTPUT
LD 2090.07  ; MASTER ON CONFIRM
IL(002)

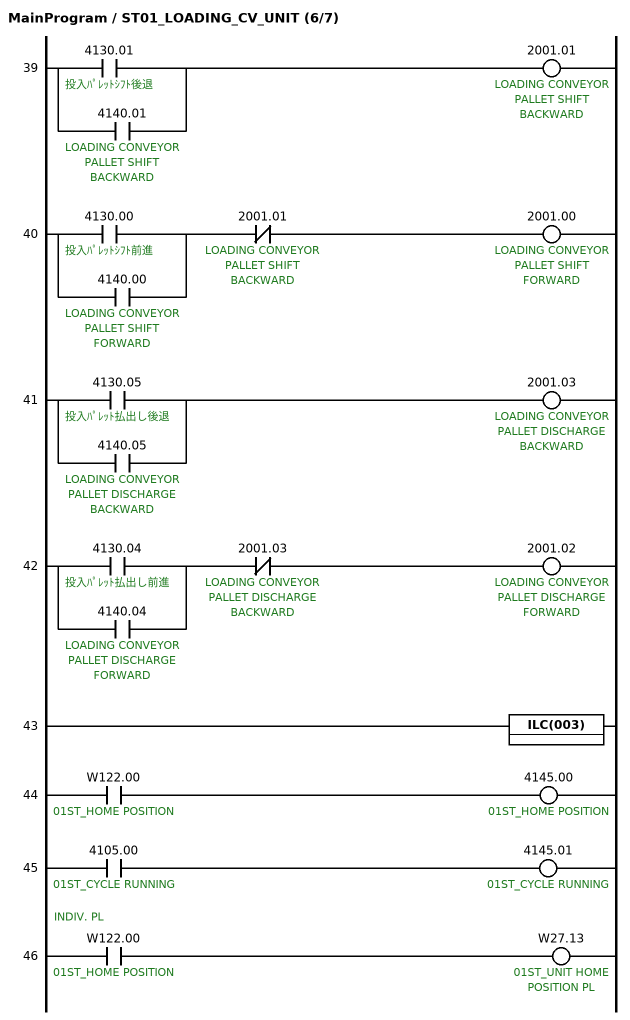
; rung 39
LD 4130.01  ; 投入ﾊﾟﾚｯﾄｼﾌﾄ後退
OR 4140.01  ; LOADING CONVEYOR PALLET SHIFT BACKWARD
OUT 2001.01  ; LOADING CONVEYOR PALLET SHIFT BACKWARD
; rung 40
LD 4130.00  ; 投入ﾊﾟﾚｯﾄｼﾌﾄ前進
OR 4140.00  ; LOADING CONVEYOR PALLET SHIFT FORWARD
ANDNOT 2001.01  ; LOADING CONVEYOR PALLET SHIFT BACKWARD
OUT 2001.00  ; LOADING CONVEYOR PALLET SHIFT FORWARD
; rung 41
LD 4130.05  ; 投入ﾊﾟﾚｯﾄ払出し後退
OR 4140.05  ; LOADING CONVEYOR PALLET DISCHARGE BACKWARD
OUT 2001.03  ; LOADING CONVEYOR PALLET DISCHARGE BACKWARD
; rung 42
LD 4130.04  ; 投入ﾊﾟﾚｯﾄ払出し前進
OR 4140.04  ; LOADING CONVEYOR PALLET DISCHARGE FORWARD
ANDNOT 2001.03  ; LOADING CONVEYOR PALLET DISCHARGE BACKWARD
OUT 2001.02  ; LOADING CONVEYOR PALLET DISCHARGE FORWARD
; rung 43
ILC(003)
; rung 44
LD W122.00  ; 01ST_HOME POSITION
OUT 4145.00  ; 01ST_HOME POSITION
; rung 45
LD 4105.00  ; 01ST_CYCLE RUNNING
OUT 4145.01  ; 01ST_CYCLE RUNNING
; rung 46: INDIV. PL
LD W122.00  ; 01ST_HOME POSITION
OUT W27.13  ; 01ST_UNIT HOME POSITION PL

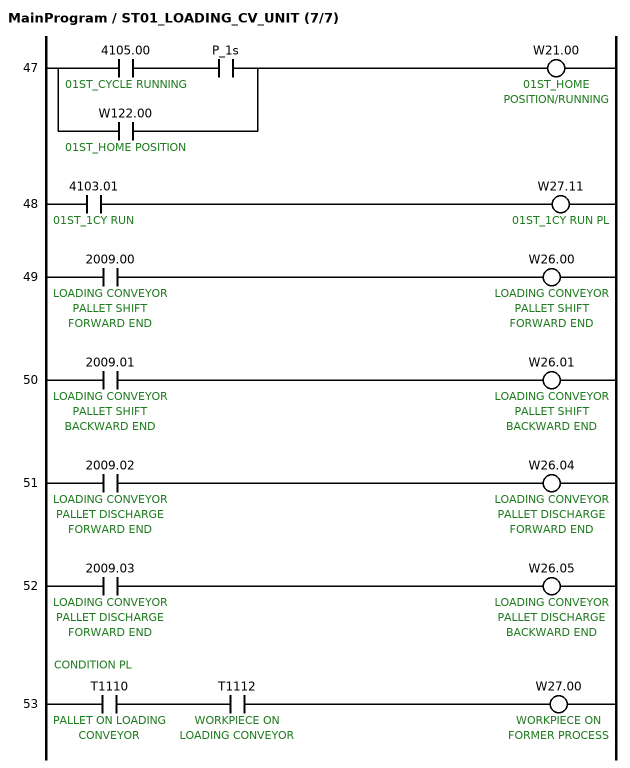
; rung 47
LD 4105.00  ; 01ST_CYCLE RUNNING
AND P_1s
OR W122.00  ; 01ST_HOME POSITION
OUT W21.00  ; 01ST_HOME POSITION/RUNNING
; rung 48
LD 4103.01  ; 01ST_1CY RUN
OUT W27.11  ; 01ST_1CY RUN PL
; rung 49
LD 2009.00  ; LOADING CONVEYOR PALLET SHIFT FORWARD END
OUT W26.00  ; LOADING CONVEYOR PALLET SHIFT FORWARD END
; rung 50
LD 2009.01  ; LOADING CONVEYOR PALLET SHIFT BACKWARD END
OUT W26.01  ; LOADING CONVEYOR PALLET SHIFT BACKWARD END
; rung 51
LD 2009.02  ; LOADING CONVEYOR PALLET DISCHARGE FORWARD END
OUT W26.04  ; LOADING CONVEYOR PALLET DISCHARGE FORWARD END
; rung 52
LD 2009.03  ; LOADING CONVEYOR PALLET DISCHARGE FORWARD END
OUT W26.05  ; LOADING CONVEYOR PALLET DISCHARGE BACKWARD END
; rung 53: CONDITION PL
LD T1110  ; PALLET ON LOADING CONVEYOR
AND T1112  ; WORKPIECE ON LOADING CONVEYOR
OUT W27.00  ; WORKPIECE ON FORMER PROCESS

### Section ST02_LOADER_UNIT
; rung 0: 02ST_LOADER UNIT

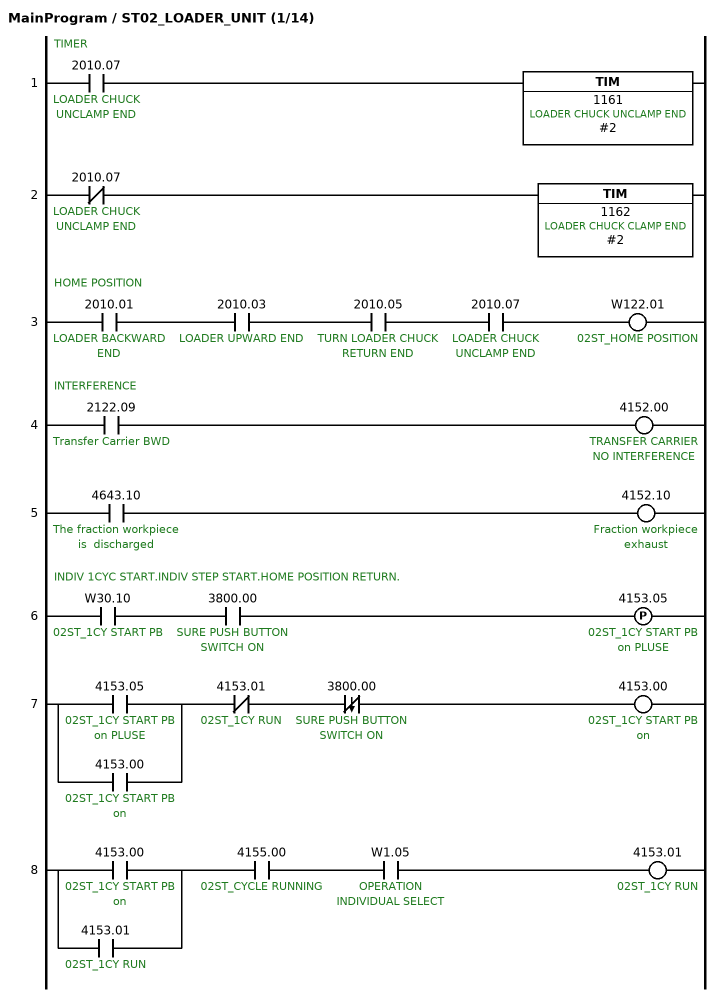
; rung 1: TIMER
LD 2010.07  ; LOADER CHUCK UNCLAMP END
TIM 1161 #2  ; LOADER CHUCK UNCLAMP END
; rung 2
LDNOT 2010.07  ; LOADER CHUCK UNCLAMP END
TIM 1162 #2  ; LOADER CHUCK CLAMP END
; rung 3: HOME POSITION
LD 2010.01  ; LOADER BACKWARD END
AND 2010.03  ; LOADER UPWARD END
AND 2010.05  ; TURN LOADER CHUCK RETURN END
AND 2010.07  ; LOADER CHUCK UNCLAMP END
OUT W122.01  ; 02ST_HOME POSITION
; rung 4: INTERFERENCE
LD 2122.09  ; Transfer Carrier BWD
OUT 4152.00  ; TRANSFER CARRIER NO INTERFERENCE
; rung 5
LD 4643.10  ; The fraction workpiece is  discharged
OUT 4152.10  ; Fraction workpiece exhaust
; rung 6: INDIV 1CYC START.INDIV STEP START.HOME POSITION RETURN.
LD W30.10  ; 02ST_1CY START PB
AND 3800.00  ; SURE PUSH BUTTON SWITCH ON
DIFU(013) 4153.05  ; 02ST_1CY START PB on PLUSE
; rung 7
LD 4153.05  ; 02ST_1CY START PB on PLUSE
OR 4153.00  ; 02ST_1CY START PB on
ANDNOT 4153.01  ; 02ST_1CY RUN
%ANDNOT 3800.00  ; SURE PUSH BUTTON SWITCH ON
OUT 4153.00  ; 02ST_1CY START PB on
; rung 8
LD 4153.00  ; 02ST_1CY START PB on
OR 4153.01  ; 02ST_1CY RUN
AND 4155.00  ; 02ST_CYCLE RUNNING
AND W1.05  ; OPERATION INDIVIDUAL SELECT
OUT 4153.01  ; 02ST_1CY RUN

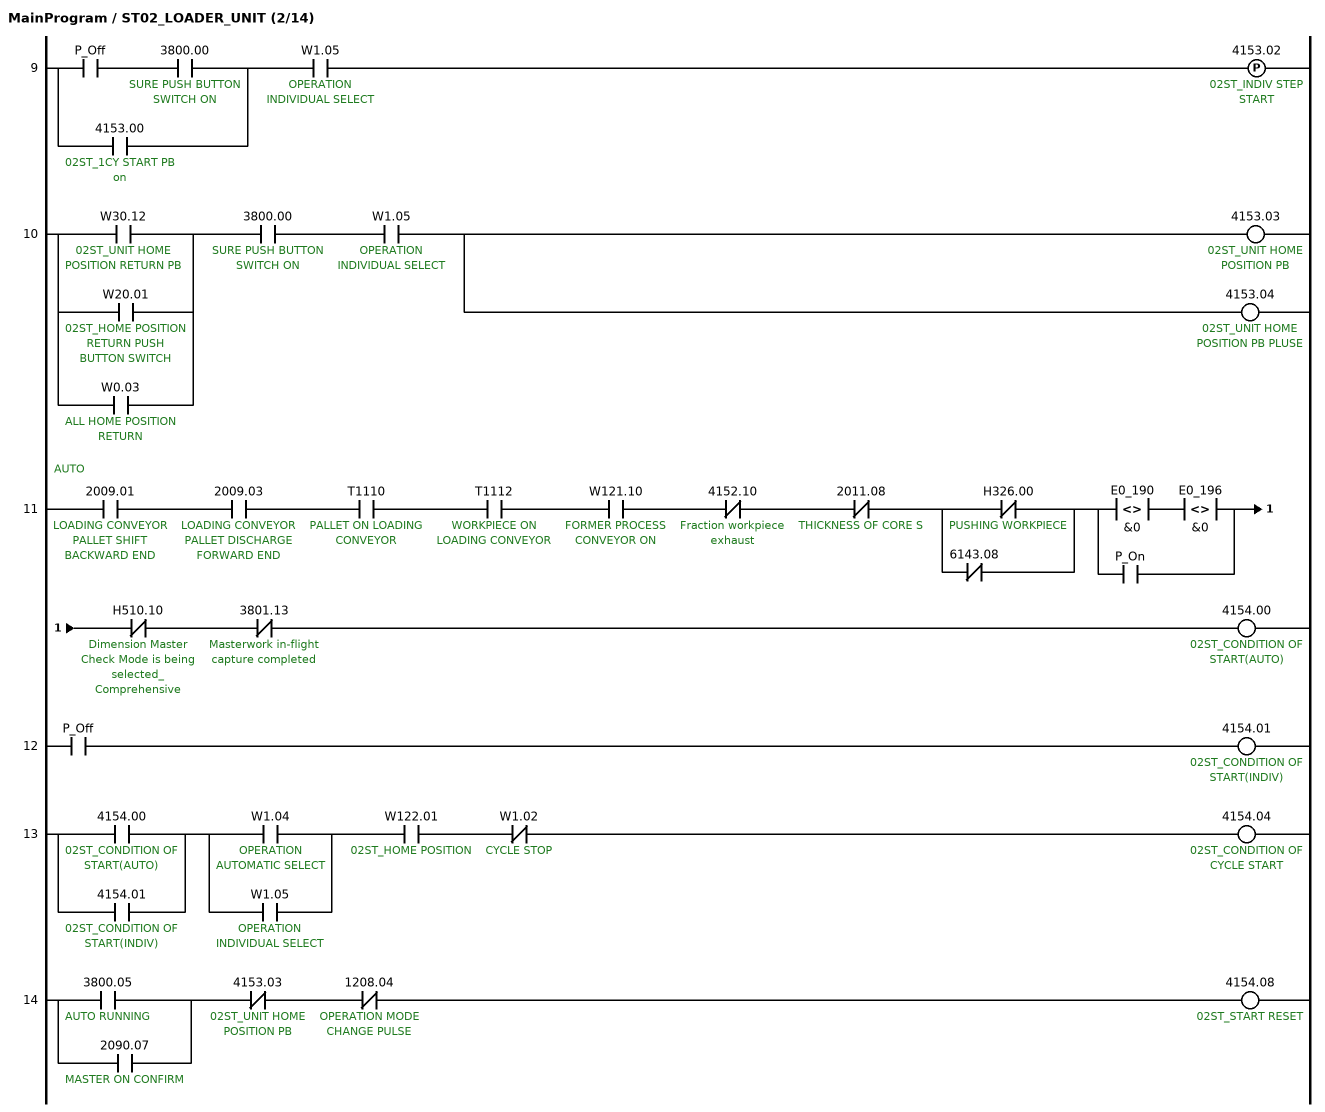
; rung 9
LD P_Off
AND 3800.00  ; SURE PUSH BUTTON SWITCH ON
OR 4153.00  ; 02ST_1CY START PB on
AND W1.05  ; OPERATION INDIVIDUAL SELECT
DIFU(013) 4153.02  ; 02ST_INDIV STEP START
; rung 10
LD W30.12  ; 02ST_UNIT HOME POSITION RETURN PB
OR W20.01  ; 02ST_HOME POSITION RETURN PUSH BUTTON SWITCH
OR W0.03  ; ALL HOME POSITION RETURN
AND 3800.00  ; SURE PUSH BUTTON SWITCH ON
AND W1.05  ; OPERATION INDIVIDUAL SELECT
OUT 4153.03  ; 02ST_UNIT HOME POSITION PB
OUT 4153.04  ; 02ST_UNIT HOME POSITION PB PLUSE
; rung 11: AUTO
LD 2009.01  ; LOADING CONVEYOR PALLET SHIFT BACKWARD END
AND 2009.03  ; LOADING CONVEYOR PALLET DISCHARGE FORWARD END
AND T1110  ; PALLET ON LOADING CONVEYOR
AND T1112  ; WORKPIECE ON LOADING CONVEYOR
AND W121.10  ; FORMER PROCESS CONVEYOR ON
ANDNOT 4152.10  ; Fraction workpiece exhaust
ANDNOT 2011.08  ; THICKNESS OF CORE S
LDNOT H326.00  ; PUSHING WORKPIECE
ORNOT 6143.08
ANDLD
LD<>(305) E0_190 &0
AND<>(305) E0_196 &0
OR P_On
ANDLD
ANDNOT H510.10  ; Dimension Master Check Mode is being selected_Comprehensive
ANDNOT 3801.13  ; Masterwork in-flight capture completed
OUT 4154.00  ; 02ST_CONDITION OF START(AUTO)
; rung 12
LD P_Off
OUT 4154.01  ; 02ST_CONDITION OF START(INDIV)
; rung 13
LD 4154.00  ; 02ST_CONDITION OF START(AUTO)
OR 4154.01  ; 02ST_CONDITION OF START(INDIV)
LD W1.04  ; OPERATION AUTOMATIC SELECT
OR W1.05  ; OPERATION INDIVIDUAL SELECT
ANDLD
AND W122.01  ; 02ST_HOME POSITION
ANDNOT W1.02  ; CYCLE STOP
OUT 4154.04  ; 02ST_CONDITION OF CYCLE START
; rung 14
LD 3800.05  ; AUTO RUNNING
OR 2090.07  ; MASTER ON CONFIRM
ANDNOT 4153.03  ; 02ST_UNIT HOME POSITION PB
ANDNOT 1208.04  ; OPERATION MODE CHANGE PULSE
OUT 4154.08  ; 02ST_START RESET

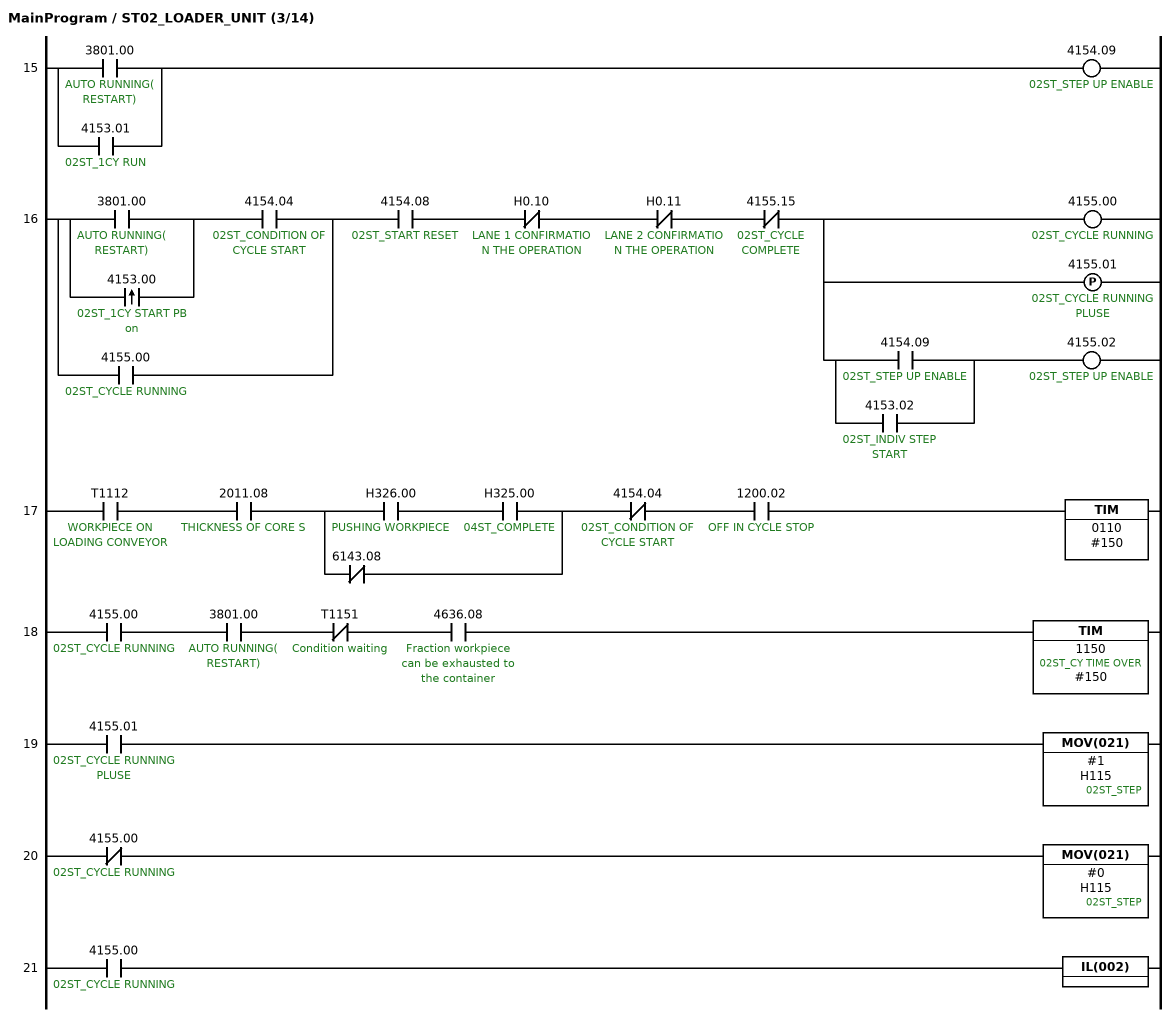
; rung 15
LD 3801.00  ; AUTO RUNNING(RESTART)
OR 4153.01  ; 02ST_1CY RUN
OUT 4154.09  ; 02ST_STEP UP ENABLE
; rung 16
LD 3801.00  ; AUTO RUNNING(RESTART)
@OR 4153.00  ; 02ST_1CY START PB on
AND 4154.04  ; 02ST_CONDITION OF CYCLE START
OR 4155.00  ; 02ST_CYCLE RUNNING
AND 4154.08  ; 02ST_START RESET
ANDNOT H0.10  ; LANE 1 CONFIRMATION THE OPERATION
ANDNOT H0.11  ; LANE 2 CONFIRMATION THE OPERATION
ANDNOT 4155.15  ; 02ST_CYCLE COMPLETE
OUT 4155.00  ; 02ST_CYCLE RUNNING
DIFU(013) 4155.01  ; 02ST_CYCLE RUNNING PLUSE
LD 4154.09  ; 02ST_STEP UP ENABLE
OR 4153.02  ; 02ST_INDIV STEP START
ANDLD
OUT 4155.02  ; 02ST_STEP UP ENABLE
; rung 17
LD T1112  ; WORKPIECE ON LOADING CONVEYOR
AND 2011.08  ; THICKNESS OF CORE S
LD H326.00  ; PUSHING WORKPIECE
AND H325.00  ; 04ST_COMPLETE
ORNOT 6143.08
ANDLD
ANDNOT 4154.04  ; 02ST_CONDITION OF CYCLE START
AND 1200.02  ; OFF IN CYCLE STOP
TIM 0110 #150
; rung 18
LD 4155.00  ; 02ST_CYCLE RUNNING
AND 3801.00  ; AUTO RUNNING(RESTART)
ANDNOT T1151  ; Condition waiting
AND 4636.08  ; Fraction workpiece can be exhausted to the container
TIM 1150 #150  ; 02ST_CY TIME OVER
; rung 19
LD 4155.01  ; 02ST_CYCLE RUNNING PLUSE
MOV(021) #1 H115  ; 02ST_STEP
; rung 20
LDNOT 4155.00  ; 02ST_CYCLE RUNNING
MOV(021) #0 H115  ; 02ST_STEP
; rung 21
LD 4155.00  ; 02ST_CYCLE RUNNING
IL(002)

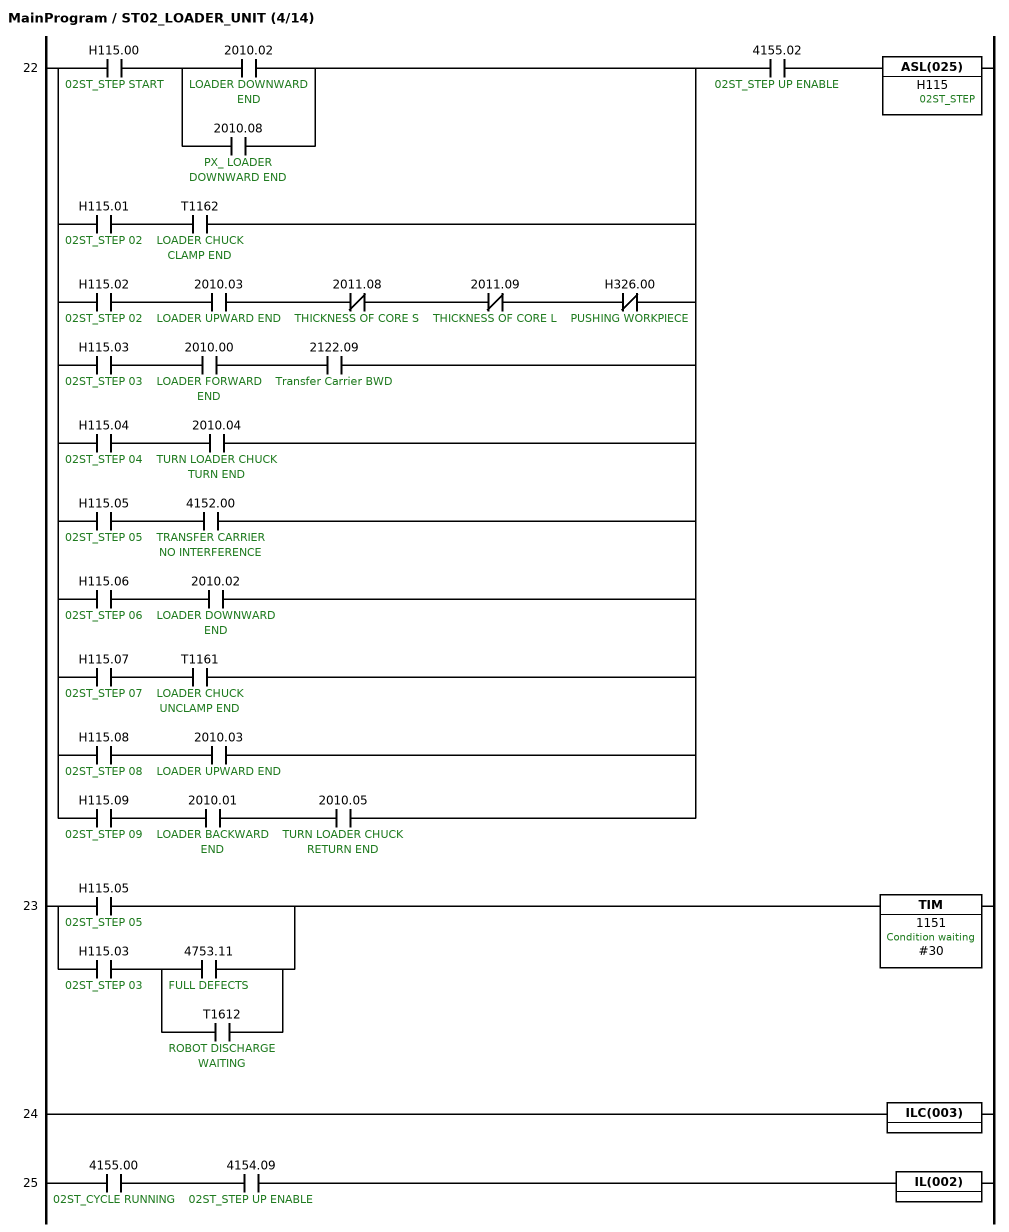
; rung 22
LD H115.00  ; 02ST_STEP START
LD 2010.02  ; LOADER DOWNWARD END
OR 2010.08  ; PX_ LOADER DOWNWARD END
ANDLD
LD H115.01  ; 02ST_STEP 02
AND T1162  ; LOADER CHUCK CLAMP END
ORLD
LD H115.02  ; 02ST_STEP 02
AND 2010.03  ; LOADER UPWARD END
ANDNOT 2011.08  ; THICKNESS OF CORE S
ANDNOT 2011.09  ; THICKNESS OF CORE L
ANDNOT H326.00  ; PUSHING WORKPIECE
ORLD
LD H115.03  ; 02ST_STEP 03
AND 2010.00  ; LOADER FORWARD END
AND 2122.09  ; Transfer Carrier BWD
ORLD
LD H115.04  ; 02ST_STEP 04
AND 2010.04  ; TURN LOADER CHUCK TURN END
ORLD
LD H115.05  ; 02ST_STEP 05
AND 4152.00  ; TRANSFER CARRIER NO INTERFERENCE
ORLD
LD H115.06  ; 02ST_STEP 06
AND 2010.02  ; LOADER DOWNWARD END
ORLD
LD H115.07  ; 02ST_STEP 07
AND T1161  ; LOADER CHUCK UNCLAMP END
ORLD
LD H115.08  ; 02ST_STEP 08
AND 2010.03  ; LOADER UPWARD END
ORLD
LD H115.09  ; 02ST_STEP 09
AND 2010.01  ; LOADER BACKWARD END
AND 2010.05  ; TURN LOADER CHUCK RETURN END
ORLD
AND 4155.02  ; 02ST_STEP UP ENABLE
ASL(025) H115  ; 02ST_STEP
; rung 23
LD H115.05  ; 02ST_STEP 05
LD H115.03  ; 02ST_STEP 03
LD 4753.11  ; FULL DEFECTS
OR T1612  ; ROBOT DISCHARGE WAITING
ANDLD
ORLD
TIM 1151 #30  ; Condition waiting
; rung 24
ILC(003)
; rung 25
LD 4155.00  ; 02ST_CYCLE RUNNING
AND 4154.09  ; 02ST_STEP UP ENABLE
IL(002)

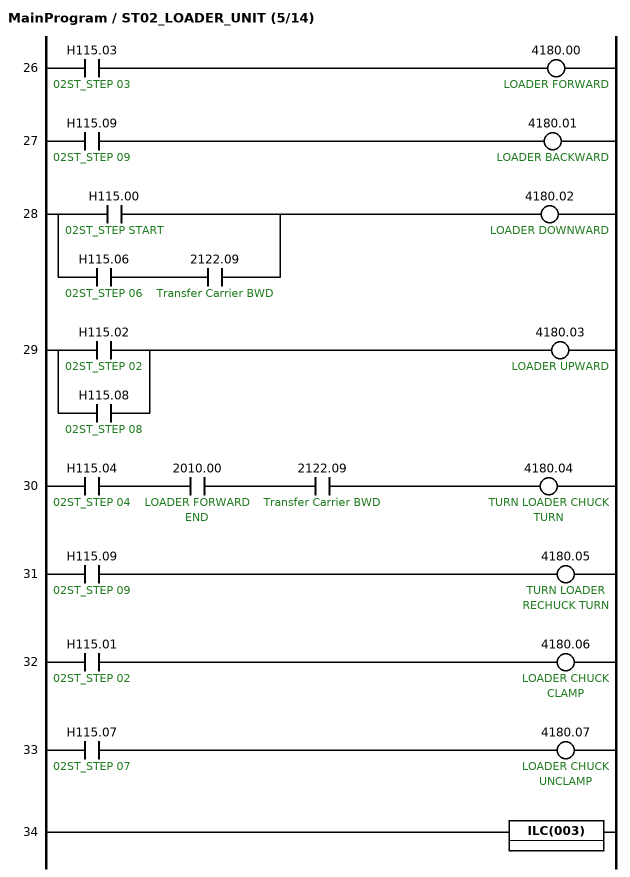
; rung 26
LD H115.03  ; 02ST_STEP 03
OUT 4180.00  ; LOADER FORWARD
; rung 27
LD H115.09  ; 02ST_STEP 09
OUT 4180.01  ; LOADER BACKWARD
; rung 28
LD H115.00  ; 02ST_STEP START
LD H115.06  ; 02ST_STEP 06
AND 2122.09  ; Transfer Carrier BWD
ORLD
OUT 4180.02  ; LOADER DOWNWARD
; rung 29
LD H115.02  ; 02ST_STEP 02
OR H115.08  ; 02ST_STEP 08
OUT 4180.03  ; LOADER UPWARD
; rung 30
LD H115.04  ; 02ST_STEP 04
AND 2010.00  ; LOADER FORWARD END
AND 2122.09  ; Transfer Carrier BWD
OUT 4180.04  ; TURN LOADER CHUCK TURN
; rung 31
LD H115.09  ; 02ST_STEP 09
OUT 4180.05  ; TURN LOADER RECHUCK TURN
; rung 32
LD H115.01  ; 02ST_STEP 02
OUT 4180.06  ; LOADER CHUCK CLAMP
; rung 33
LD H115.07  ; 02ST_STEP 07
OUT 4180.07  ; LOADER CHUCK UNCLAMP
; rung 34
ILC(003)

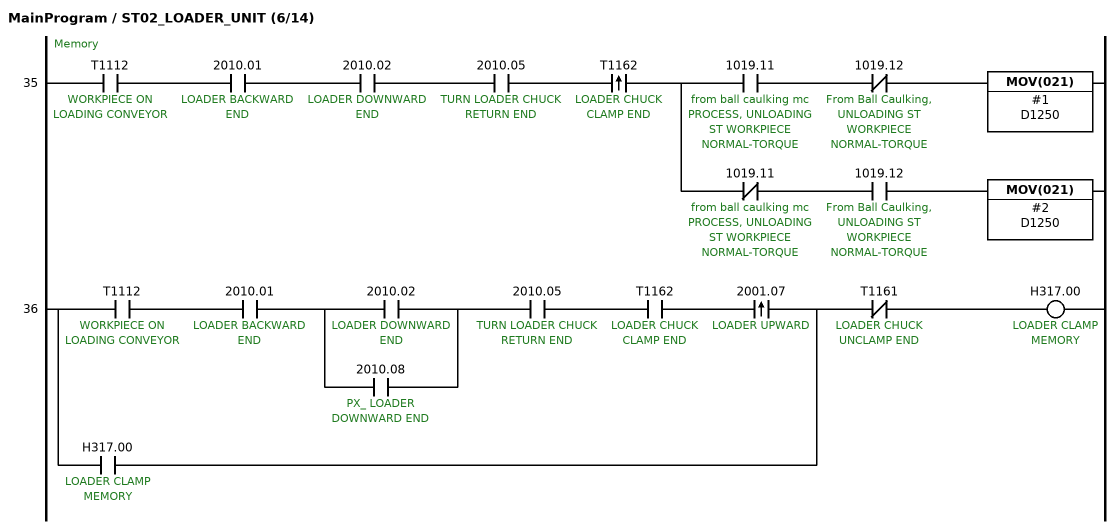
; rung 35: Memory
LD T1112  ; WORKPIECE ON LOADING CONVEYOR
AND 2010.01  ; LOADER BACKWARD END
AND 2010.02  ; LOADER DOWNWARD END
AND 2010.05  ; TURN LOADER CHUCK RETURN END
@AND T1162  ; LOADER CHUCK CLAMP END
OUT TR0
AND 1019.11  ; from ball caulking mc  PROCESS, UNLOADING ST WORKPIECE NORMAL-TORQUE
ANDNOT 1019.12  ; From Ball Caulking, UNLOADING ST WORKPIECE NORMAL-TORQUE
MOV(021) #1 D1250
LD TR0
ANDNOT 1019.11  ; from ball caulking mc  PROCESS, UNLOADING ST WORKPIECE NORMAL-TORQUE
AND 1019.12  ; From Ball Caulking, UNLOADING ST WORKPIECE NORMAL-TORQUE
MOV(021) #2 D1250
; rung 36
LD T1112  ; WORKPIECE ON LOADING CONVEYOR
AND 2010.01  ; LOADER BACKWARD END
LD 2010.02  ; LOADER DOWNWARD END
OR 2010.08  ; PX_ LOADER DOWNWARD END
ANDLD
AND 2010.05  ; TURN LOADER CHUCK RETURN END
AND T1162  ; LOADER CHUCK CLAMP END
@AND 2001.07  ; LOADER UPWARD
OR H317.00  ; LOADER CLAMP MEMORY
ANDNOT T1161  ; LOADER CHUCK UNCLAMP END
OUT H317.00  ; LOADER CLAMP MEMORY

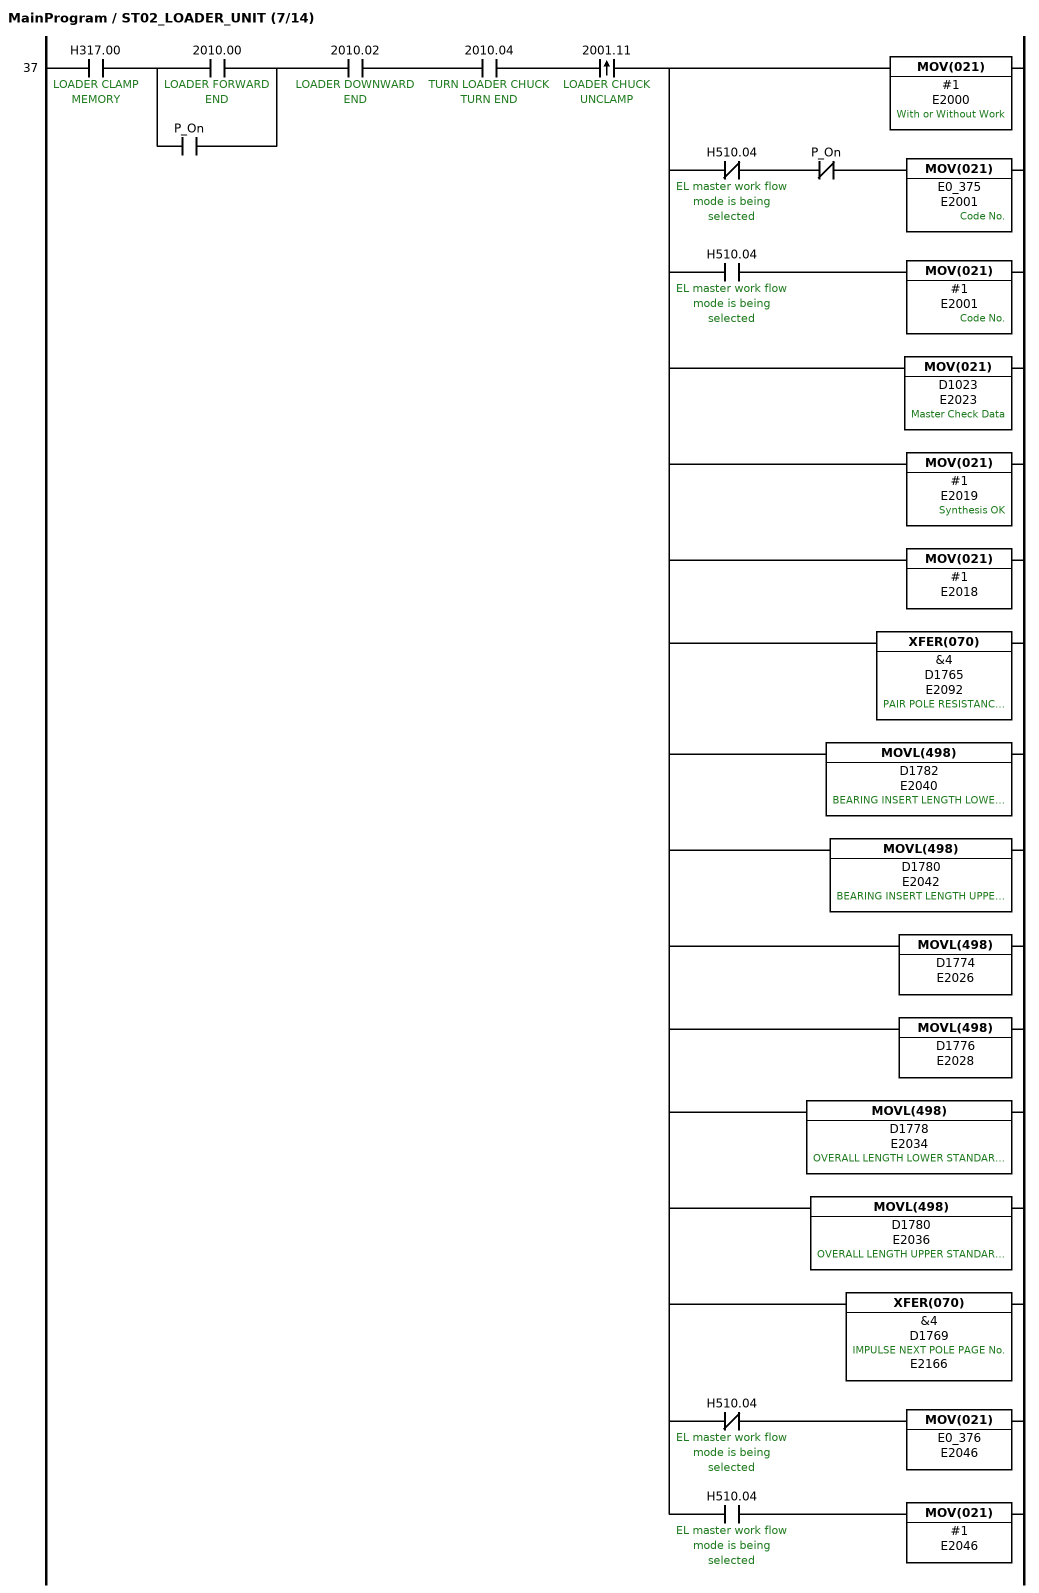
; rung 37
LD H317.00  ; LOADER CLAMP MEMORY
LD 2010.00  ; LOADER FORWARD END
OR P_On
ANDLD
AND 2010.02  ; LOADER DOWNWARD END
AND 2010.04  ; TURN LOADER CHUCK TURN END
@AND 2001.11  ; LOADER CHUCK UNCLAMP
OUT TR0
MOV(021) #1 E2000  ; With or Without Work
ANDNOT H510.04  ; EL master work flow mode is being selected
ANDNOT P_On
MOV(021) E0_375 E2001  ; Code No.
LD TR0
AND H510.04  ; EL master work flow mode is being selected
MOV(021) #1 E2001  ; Code No.
LD TR0
MOV(021) D1023 E2023  ; Master Check Data
MOV(021) #1 E2019  ; Synthesis OK
MOV(021) #1 E2018
XFER(070) &4 D1765 E2092  ; PAIR POLE RESISTANCE SPECIFICATION MINIMUM VALUE
MOVL(498) D1782 E2040  ; BEARING INSERT LENGTH LOWER STANDARD VALUE
MOVL(498) D1780 E2042  ; BEARING INSERT LENGTH UPPER STANDARD VALUE
MOVL(498) D1774 E2026
MOVL(498) D1776 E2028
MOVL(498) D1778 E2034  ; OVERALL LENGTH LOWER STANDARD VALUE
MOVL(498) D1780 E2036  ; OVERALL LENGTH UPPER STANDARD VALUE
XFER(070) &4 D1769 E2166  ; IMPULSE NEXT POLE PAGE No.
ANDNOT H510.04  ; EL master work flow mode is being selected
MOV(021) E0_376 E2046
LD TR0
AND H510.04  ; EL master work flow mode is being selected
MOV(021) #1 E2046

